// TwinCAT 3 PLC project CNC
// ProgramVersion: 3.1.4020.2
// libraries:
//   Tc2_ControllerToolbox, * (Beckhoff Automation GmbH)
//   Tc2_MC2, * (Beckhoff Automation GmbH)
//   Tc2_Standard, * (Beckhoff Automation GmbH)
//   Tc2_System, * (Beckhoff Automation GmbH)
//   Tc2_TcpIp, * (Beckhoff Automation GmbH)
//   Tc3_Interfaces, * (Beckhoff Automation GmbH)
//   Tc3_Module, * (Beckhoff Automation GmbH)
//   VisuDialogs, * (System)
// project tree:
//   DUTs/ E_ModeMMA.TcDUT, ST_Param.TcDUT, ST_ParamFixed.TcDUT, ST_ParamMachine.TcDUT, ST_ParamRecipe.TcDUT, ST_ParamStatus.TcDUT
//   DUTs/Param/ ST_Palette.TcDUT, ST_Position.TcDUT
//   / ErrorList.TcTLO, GlobalImagePool.TcGIPO (not stored), GlobalTextList.TcGTLO, PlcTask.TcTTO, Visualisierungsmanager.TcVMO (not stored), VISU_TASK.TcTTO
//   FB_Lib/Conversion/ FB_ConfigAnalog.TcPOU, FB_Ia.TcPOU, FB_Qa.TcPOU, ST_MinMax.TcDUT
//   FB_Lib/FB_ActionneurSimple/ FB_ActionneurSimple.TcPOU, ST_Erreur.TcDUT, ST_ParamActionneur.TcDUT
//   FB_Lib/ FB_Etape.TcPOU, FB_RegulMoteur.TcPOU (excluded from build)
//   FB_Lib/FB_GestionModes/ FB_Btn.TcPOU, FB_CycleAuto.TcPOU, FB_CycleInit.TcPOU, FB_CycleMan.TcPOU, FB_MMA.TcPOU, p_InitVar.TcPOU
//   FB_Lib/FB_GestionModes/IO/ ST_IO.TcDUT, ST_IOInput.TcDUT, ST_IOInputSimul.TcDUT, ST_IOOutput.TcDUT, ST_IOOutputSimul.TcDUT
//   FB_Lib/Motor/ FB_Moteur.TcPOU, ST_ParamMoteur.TcDUT, ST_ParamMoveMoteur.TcDUT
//   FB_Lib/TCPIP/ FB_TCP.TcPOU, ST_Output.TcDUT, ST_ParamTCP.TcDUT, ST_TxRx.TcDUT
//   GVLs/ GVL.TcGVL
//   POUs/ MAIN.TcPOU
//   VISUs/ Visu2_MainCtr.TcVIS, Visu2_LanguageUser.TcVIS, Visu2_Status.TcVIS, Visu2_StatusSimple.TcVIS, VisuAdmin.TcVIS, Visualization.TcVIS, VisuAuto.TcVIS, VisuInit.TcVIS, VisuManual.TcVIS, VisuMMA.TcVIS, VisuMotor.TcVIS (excluded from build)
// real-time tasks:
//   TASK PlcTask: cycle T#10ms, priority 10, ADS port 351
//   TASK VISU_TASK: cycle T#50000us, priority 12, ADS port 350
// motion (NC):
//   TASK NC-Task 1 SAF: cycle T#2ms, priority 4, ADS port 501
//   TASK NC-Task 1 SVB: cycle T#10ms, priority 8, ADS port 511
//   AXIS Axis 1 (id 1)
//     Dynamic: Acceleration=60900.1, Deceleration=60900.1, Jerk=1431970
//     Velo: RefSync=10, SlowManual=25, FastManual=3500, Maximum=3500
//     OtherSettings: AllowMotionCmdToSlave=true
//     encoder EncType=25
//       EncPara: ScaleFactorNumerator=360, ScaleFactorDenominator=12800, MaxCount=#x0000ffff
//         SoftEndMinControl: Enable=true
//         SoftEndMaxControl: Enable=true, Range=5000
//     drive DrvType=20
//       Analog: VeloReferenz=3500
//       TimeComp: TaskDelayCycles=1
//     controller CtrType=1
//       CtrPara: PriorControlFactor=1
//         PosDiffControl: Enable=false
//         PID: PosKp=60
//         Observer: BandWidth=20
//   AXIS Achse 2 - Y (id 2)
//     General: UnitName=°
//     Dynamic: Acceleration=127260, Deceleration=127260, Jerk=25706400
//     Velo: RefSearch=500, RefSync=100, SlowManual=20, FastManual=40000, Maximum=58000
//     TargetPosControl: Range=10
//     OtherSettings: AllowMotionCmdToSlave=true
//     encoder EncType=26
//       EncPara: ScaleFactorNumerator=360, ScaleFactorDenominator=2048, MaxCount=#x0000ffff
//         SoftEndMinControl: Enable=true
//         SoftEndMaxControl: Enable=true, Range=5000
//     drive DrvType=21
//       Analog: VeloReferenz=58000
//       TimeComp: TaskDelayCycles=1
//     controller CtrType=3
//       CtrPara: PriorControlFactor=1
//         PosDiffControl: Enable=false
//         PID: PosKp=30, PosTn=0.2, PosTv=0.2, PosTd=0.2, PosIOutputLimit=0.25, PosDOutputLimit=0.25
//         Observer: BandWidth=20
//   AXIS Achse 3 - Z (id 3)
//     Dynamic: Acceleration=3611.11, Deceleration=3611.11, Jerk=117362
//     Velo: Maximum=3500
//     OtherSettings: AllowMotionCmdToSlave=true
//     encoder EncType=1
//       EncPara: ScaleFactorNumerator=360, ScaleFactorDenominator=12600
//         SoftEndMinControl: Enable=true
//         SoftEndMaxControl: Enable=true, Range=125
//     drive DrvType=5
//       Analog: VeloReferenz=3500
//       TimeComp: TaskDelayCycles=1
//     controller CtrType=1
//       CtrPara: PriorControlFactor=1
//         PosDiffControl: Enable=false
//         PID: PosKp=60
//         Observer: BandWidth=20
// I/O:
//   DEVICE Gerät 2 (EtherCAT)
//     Box 1 (BK1150)
//     Box 2 (BK1150) (disabled)
// variable links:
//   NC-Task 1 SAF/Axes/Achse 2 - Y <-> Device 2 (EtherCAT)/Box 1 (BK1150)
//     Drive/Inputs/In/nState1 @bit 4 <-> Term 4 (KL2552)/Channel 1/Status @bit 4
//     Drive/Outputs/Out/nCtrl1 @bit 5 <-> Term 4 (KL2552)/Channel 1/Kontrolle @bit 5
//     Drive/Outputs/Out/nDataOut2[0] <-> Term 4 (KL2552)/Channel 1/Daten Aus
//     Enc/Inputs/In/nDataIn1[0] <-> Term 4 (KL2552)/Channel 1/Daten Ein
//     Enc/Inputs/In/nState1 @bit 2 <-> Term 4 (KL2552)/Channel 1/Status
//     Enc/Outputs/Out/nCtrl1 @bit 1 <-> Term 4 (KL2552)/Channel 1/Kontrolle
//   NC-Task 1 SAF/Axes/Axis 1 <-> Device 2 (EtherCAT)/Box 1 (BK1150)
//     Drive/Inputs/In/nState1 <-> Term 3 (KL2531)/Channel 1/Status
//     Drive/Outputs/Out/nCtrl1 <-> Term 3 (KL2531)/Channel 1/Ctrl
//     Drive/Outputs/Out/nDataOut2[0] <-> Term 3 (KL2531)/Channel 1/Velocity
//     Enc/Inputs/In/nDataIn1[0] <-> Term 3 (KL2531)/Channel 1/Position
//     Enc/Inputs/In/nState1 <-> Term 3 (KL2531)/Channel 1/ExtStatus
//     Enc/Outputs/Out/nCtrl1 <-> Term 3 (KL2531)/Channel 1/ExtCtrl
//   CNC/CNC Instance <-> Device 2 (EtherCAT)/Box 1 (BK1150)
//     PlcTask Inputs/GVL.fbAct1.IxSensIn <-> Term 7 (KL1408)/Channel 2/Eingang
//     PlcTask Inputs/GVL.fbAct1.IxSensOut <-> Term 7 (KL1408)/Channel 1/Eingang
//     PlcTask Inputs/GVL.stIO.stIn.IxAruIO <-> Term 8 (KL1408)/Channel 1/Eingang
//     PlcTask Inputs/GVL.stIO.stIn.xAirPressureOk <-> Term 8 (KL1408)/Channel 4/Eingang
//     PlcTask Inputs/GVL.stIO.stIn.xAllowedGetPiece <-> Term 7 (KL1408)/Channel 6/Eingang
//     PlcTask Inputs/GVL.stIO.stIn.xPiecePresent <-> Term 7 (KL1408)/Channel 7/Eingang
//     PlcTask Outputs/GVL.fbAct1.QxBlockingValve <-> Term 10 (KL2408)/Channel 2/Ausgang
//     PlcTask Outputs/GVL.fbAct1.QxInOutput <-> Term 9 (KL2408)/Channel 6/Ausgang
//     PlcTask Outputs/GVL.fbAct1.QxOutOutput <-> Term 9 (KL2408)/Channel 5/Ausgang
//     PlcTask Outputs/GVL.stIO.stOut.QxLampeOrange <-> Term 9 (KL2408)/Channel 2/Ausgang
//     PlcTask Outputs/GVL.stIO.stOut.QxLampeRed <-> Term 9 (KL2408)/Channel 1/Ausgang
//     PlcTask Outputs/GVL.stIO.stOut.QxLampeVerte <-> Term 9 (KL2408)/Channel 3/Ausgang
//   CNC/CNC Instance <-> NC-Task 1 SAF/Axes/Achse 2 - Y
//     PlcTask Inputs/GVL.fbMotorY.fbAxisRef.NcToPlc <-> Outputs/ToPlc
//     PlcTask Outputs/GVL.fbMotorY.fbAxisRef.PlcToNc <-> Inputs/FromPlc
//   CNC/CNC Instance <-> NC-Task 1 SAF/Axes/Achse 3 - Z
//     PlcTask Inputs/GVL.fbMotorZ.fbAxisRef.NcToPlc <-> Outputs/ToPlc
//     PlcTask Outputs/GVL.fbMotorZ.fbAxisRef.PlcToNc <-> Inputs/FromPlc
//   CNC/CNC Instance <-> NC-Task 1 SAF/Axes/Axis 1
//     PlcTask Inputs/GVL.fbMotorX.fbAxisRef.NcToPlc <-> Outputs/ToPlc
//     PlcTask Outputs/GVL.fbMotorX.fbAxisRef.PlcToNc <-> Inputs/FromPlc

CONFIGURATION CNC
    RESOURCE PLC ON TwinCAT3
        TASK PlcTask(INTERVAL := T#10ms, PRIORITY := 10);
        TASK VISU_TASK(INTERVAL := T#50000us, PRIORITY := 12);
        PROGRAM MAIN WITH PlcTask : MAIN;
        PROGRAM VisuElems_Visu_Prg WITH VISU_TASK : VisuElems.Visu_Prg;
    END_RESOURCE
END_CONFIGURATION

// ---- DUTs/E_ModeMMA.TcDUT

TYPE E_ModeMMA :
(
	Init := 0,
	Auto,
	Man
);
END_TYPE

// ---- DUTs/Param/ST_Palette.TcDUT
TYPE ST_Palette :
STRUCT
	PaletteDimensionX : INT;
	PaletteDimensionY : INT;
	
	ActualPalettePositionX : INT;
	ActualPalettePositionY : INT;
END_STRUCT
END_TYPE

// ---- DUTs/Param/ST_Position.TcDUT
TYPE ST_Position :
STRUCT
	PosX : LREAL;
	PosY: LREAL;
	Initialized: BOOL;
END_STRUCT
END_TYPE

// ---- DUTs/ST_Param.TcDUT
TYPE ST_Param :
STRUCT
	stStatus:ST_ParamStatus;	//informations d'états (compteur de pièces, modes,...)
	stFixed:ST_ParamFixed;		//Paramètres pas en lien avec le produit, fixe
	stRecipe:ST_ParamRecipe;	//Paramètres en lien avec le produit
	stMachine:ST_ParamMachine;	//Parametres de la machine
END_STRUCT
END_TYPE

// ---- DUTs/ST_ParamFixed.TcDUT
TYPE ST_ParamFixed :
STRUCT
END_STRUCT
END_TYPE

// ---- DUTs/ST_ParamMachine.TcDUT
TYPE ST_ParamMachine :
STRUCT
	stParamMotX:ST_ParamMoteur;		//parametres des trois Moteurs
	stParamMotY:ST_ParamMoteur;
	stParamMotZ:ST_ParamMoteur;
	
	stPosition0: ST_Position;		//Position Home
	stPosition1: ST_Position;		//Position Palette bottom left
	stPosition2: ST_Position;		//Position Palette bottom right
	stPosition3: ST_Position;		//Position Palette top left
	stPosition4: ST_Position;		//Position Prise Piece


END_STRUCT
END_TYPE

// ---- DUTs/ST_ParamRecipe.TcDUT
TYPE ST_ParamRecipe :
STRUCT
	stPalette1 : ST_Palette;
END_STRUCT
END_TYPE

// ---- DUTs/ST_ParamStatus.TcDUT
TYPE ST_ParamStatus :
STRUCT
	eMMA : E_ModeMMA; 
	xModePasAPas:BOOL;
	xErreur:BOOL;		//shows the current error state
	iId : INT; 			//error number currently active
	sMessage : STRING; 	//error message for the active error
	xInitOk:BOOL;		//indique que l'initialisation a été exécutée
	xHomingDone : BOOL;	//indique q'on a fait un homing depuis la derniere mise en puissance
END_STRUCT
END_TYPE

// ---- FB_Lib/Conversion/ST_MinMax.TcDUT
TYPE ST_MinMax :
STRUCT
	lrMin: LREAL;
	lrMax: LREAL;
END_STRUCT
END_TYPE

// ---- FB_Lib/FB_ActionneurSimple/ST_Erreur.TcDUT
TYPE ST_Erreur :
STRUCT
	xState:BOOL; 		//shows the current error state
	iId : INT; 			//error number currently active
END_STRUCT
END_TYPE

// ---- FB_Lib/FB_ActionneurSimple/ST_ParamActionneur.TcDUT
TYPE ST_ParamActionneur :
STRUCT
	tTimeOut : TIME; 			//max time allowed for moving to position bevor xState=TRUE
	xPresenceSensOut : BOOL; 	//If at the out-pos a Sensor is available
	xPresenceSensIn : BOOL; 	//If at the in-pos a Sensor is availaible
	tMoveOutTimeDelay : TIME; 	//delay after activating xPresenceSensOut before turning off output. When there is no Sensor, only this time will be used.
	tMoveInTimeDelay : TIME; 	//delay after activating xPresenceSensIn before turning off output. When there is no Sensor, only this time will be used.
END_STRUCT
END_TYPE

// ---- FB_Lib/FB_GestionModes/IO/ST_IO.TcDUT
TYPE ST_IO :
STRUCT
	stIn:ST_IOInput;
	stOut:ST_IOOutput;
END_STRUCT
END_TYPE

// ---- FB_Lib/FB_GestionModes/IO/ST_IOInput.TcDUT
TYPE ST_IOInput :
STRUCT
	IxAruIO AT%I*  :BOOL;
	xStartIO AT%I* :BOOL;
	xStopIO AT%I*  :BOOL;
	xResetIO AT%I* :BOOL;
	xAuto AT%I* : BOOL;
	xManual AT%I* : BOOL;
	
	
	
	iSetSpeedMotor : INT := 10;
	
	xAirPressureOk AT%I* : BOOL;
	
	//Btn in manual mode
	xHomingPosReached AT%I* : BOOL;
	xManualAct1GoIn AT%I* : BOOL;
	xManualAct1GoOut AT%I* : BOOL;
	
	//Btn in init mode
	xSetHomePos   AT%I*: BOOL;
	xJogXForward  AT%I*: BOOL;
	xJogYForward  AT%I*: BOOL;
	xJogXBackward AT%I*: BOOL;
	xJogYBackward AT%I*: BOOL;
	
	//Auto mode
	xAllowedGetPiece AT%I* : BOOL;
	xPiecePresent AT%I* : BOOL;
	xEmulateZDone AT%I* :Bool;
	
END_STRUCT
END_TYPE

// ---- FB_Lib/FB_GestionModes/IO/ST_IOInputSimul.TcDUT
TYPE ST_IOInputSimul :
STRUCT
	IxAru :BOOL;
END_STRUCT
END_TYPE

// ---- FB_Lib/FB_GestionModes/IO/ST_IOOutput.TcDUT
TYPE ST_IOOutput :
STRUCT
	QxLampeRed AT%Q*:BOOL;
	QxLampeVerte AT%Q* : BOOL;
	QxLampeOrange AT%Q* :BOOL;
	
	
END_STRUCT
END_TYPE

// ---- FB_Lib/FB_GestionModes/IO/ST_IOOutputSimul.TcDUT
TYPE ST_IOOutputSimul :
STRUCT
	QxLampeRed AT%Q*:BOOL;
END_STRUCT
END_TYPE

// ---- FB_Lib/Motor/ST_ParamMoteur.TcDUT
TYPE ST_ParamMoteur :
STRUCT
	stMoveLent:ST_ParamMoveMoteur;//paramètre déplacement lent
	stMoveRapide:ST_ParamMoveMoteur;//paramètre déplacement rapide
	lrPositionInitiale:LREAL:=0;//valeur de position initiale après un MC_Home;
	mcHomingMode:MC_HomingMode:=MC_Direct;//type homing
	(*HomingMode determines in which way the calibration is carried out.
    MC_DefaultHoming
    Initiates standard homing.
    MC_Direct
    Sets the axis position directly to Position without executing a movement.
    MC_ForceCalibration
    Enforces the "axis is calibrated" state. No movement takes place, and the position remains unchanged.
    MC_ResetCalibration
    Resets the calibration state of the axis. No movement takes place, and the position remains unchanged.*)
END_STRUCT
END_TYPE

// ---- FB_Lib/Motor/ST_ParamMoveMoteur.TcDUT
TYPE ST_ParamMoveMoteur :
STRUCT
	lrVitesse:LREAL:=900;			//vitesse
	lrAcceleration:LREAL:=0;		//accélération standard, 0 si standard
	lrDecceleration:LREAL:=0;		//accélération standard, 0 si standard
END_STRUCT
END_TYPE

// ---- FB_Lib/TCPIP/ST_Output.TcDUT
TYPE ST_Output :
STRUCT
	xBusy: BOOL;
	xError: BOOL;
	nErrID : INT;
	Resulte : STRING;
	Resulth : STRING;
	Resultd : STRING;
	Boole : INT;
	Boolh : INT;
	Boold : INT;
END_STRUCT
END_TYPE

// ---- FB_Lib/TCPIP/ST_ParamTCP.TcDUT
TYPE ST_ParamTCP :
STRUCT
	sRemoteHost : T_IPV4Addr;
	nRemotePort : UDINT;
	tTimeout: TIME;
	xConnected : BOOL;			//TRUE if currently Connected to a Server
	hSocket : T_HSOCKET;		//saves the connection details after the first Connection
	xCognexMode : BOOL;			//login in into an cognex Camera
	sCognexUser: STRING;
	sCognexPW: STRING;
	xConnectedCognex: BOOL;		//connection to Cognex etablished
	NetID :  T_AmsNetId;
END_STRUCT
END_TYPE

// ---- FB_Lib/TCPIP/ST_TxRx.TcDUT
TYPE ST_TxRx :
STRUCT
	sSend : STRING;
	sReceived: STRING;
END_STRUCT
END_TYPE

// ---- GVLs/GVL.TcGVL
VAR_GLOBAL

	fbAct1:FB_ActionneurSimple;	//Act1 corresponds to holding the object
	
	xModeStepForStep :BOOL;
	xNextStep : BOOL;
	
	//pour FB_gestion du mode
	fbMMA:FB_MMA;
	fbCycleAuto:FB_CycleAuto;
	fbCycleInit : FB_CycleInit;
	fbCycleMan : FB_CycleMan;
	
	stParam:ST_Param;
	fbBtn:FB_Btn;
	stIO:ST_IO;
	
	//Tachymetre moteur
	//fbMotor : FB_RegulMoteur;
	fbMotorX : FB_Moteur;
	fbMotorY : FB_Moteur;
	fbMotorZ : FB_Moteur;
	

	 
END_VAR

// ---- POUs/MAIN.TcPOU
PROGRAM MAIN
VAR
END_VAR

//******************************************
//cyclic call of all needed FB
//******************************************
ACT_Moteur();
ACT_Actor();

fbMMA();

//copy physical Inputs in fbBtn
fbBtn.xAru:=stio.stIn.IxAruIO;
fbBtn.xReset:=stio.stIn.xResetIO OR NOT stio.stIn.xAirPressureOk;
fbBtn.xStart:=stio.stIn.xStartIO;
fbBtn.xStop:=stio.stIn.xStopIO;
fbBtn.xAirPressureOk:=stio.stIn.xAirPressureOk;
fbBtn.xManualAct1GoIn:=stio.stIn.xManualAct1GoIn;
fbBtn.xManualAct1GoOut:=stio.stIn.xManualAct1GoOut;
fbBtn.xHomingPosReached:=stio.stIn.xHomingPosReached;
fbBtn.xSetHomePos:=stio.stIn.xSetHomePos;
fbBtn.xAllowedGetPiece:=stio.stIn.xAllowedGetPiece;
fbBtn.xPiecePresent:=stio.stIn.xPiecePresent;
fbBtn.xEmulateZDone:=stio.stIn.xEmulateZDone;
fbBtn.xJogXBackward:=stio.stIn.xJogXBackward;
fbBtn.xJogYBackward:=stio.stIn.xJogYBackward;
fbBtn.xJogXForward:=stio.stIn.xJogXForward;
fbBtn.xJogYForward:=stio.stIn.xJogYForward;
fbBtn.iMotorSpeed:=stio.stIn.iSetSpeedMotor;


//and now call it
fbBtn();

//stParam
//check for active errors
IF (fbAct1.stError.xState) THEN
	stParam.stStatus.xErreur:=TRUE;
	stParam.stStatus.iId:=fbAct1.stError.iId;
ELSIF (fbCycleAuto.xError) THEN
	stParam.stStatus.xErreur:=TRUE;
	stParam.stStatus.iId:=fbCycleAuto.iId;
ELSIF NOT fbBtn.xAirPressureOk THEN
	stParam.stStatus.xErreur:=TRUE;
	stParam.stStatus.iId:=1;
ELSE
	//clear the error State. Do not clear the last error Message to have some kind of error history
	stParam.stStatus.xErreur:=FALSE;
END_IF

//call auto mode and give over the needed parameters
fbCycleAuto.xStart:=fbMMA.iEtape=350;
fbCycleAuto.xStop:= fbMMA.iEtape=390;
fbCycleAuto.xReset:= fbMMA.iEtape=810 OR fbMMA.iEtape=910;
fbCycleAuto();

//call Init mode and give over the needed parameters
fbCycleInit.xStart:=(fbMMA.iEtape=110 OR fbMMA.iEtape=340);
fbCycleInit.xStop:= NOT (fbMMA.iEtape=111 OR fbMMA.iEtape=341);
fbCycleInit.xReset:= fbMMA.iEtape=810 OR fbMMA.iEtape=910;
fbCycleInit();
	
//call Manual mode and give over the needed parameters
fbCycleMan.xStart:= fbMMA.iEtape=210;
fbCycleMan.xStop:=  fbMMa.iEtape<>210;
fbCycleMan();


//******************************************
//Output actions
//******************************************

//activate Lamp1
stIo.stOut.QxLampeRed:=NOT fbBtn.xAru;

ACTION ACT_Actor:
//Air-Actor controlling part
//cyclic call of the FB-blocs
fbAct1();	//Act2 corresponds to taking the object

//actuator movement autorize only if not in ARU
fbAct1.xAutorizeIn:=fbBtn.xAru;
fbAct1.xAutorizeOut:=fbBtn.xAru;

//move in and out each actuator
fbAct1.xInGoOut:=fbCycleAuto.iEtape=113 OR fbCycleMan.iEtape=202;

fbAct1.xInGoIn:=fbCycleAuto.iEtape=180 OR fbCycleAuto.iEtape=122 OR fbCycleAuto.iEtape=150 OR fbCycleAuto.iEtape=800 OR fbCycleInit.iEtape=400 OR fbCycleMan.iEtape=201;

//Reset des Actionneurs avan le init
fbAct1.xReset:=fbCycleInit.iEtape=99 OR fbMMA.iEtape=810;
END_ACTION

ACTION ACT_Moteur:
//Motor controlling part
//exécution de l'appel du bloc moteur
fbMotorX(stParam:=stParam.stMachine.stParamMotX);
fbMotorY(stParam:=stParam.stMachine.stParamMotY);
fbMotorZ(stParam:=stParam.stMachine.stParamMotZ);


//pilotage mise en puissance
fbMotorX.mcPower.Enable:=stIO.stIn.IxAruIO;
fbMotorX.mcPower.Enable_Negative:=stIO.stIn.IxAruIO;
fbMotorX.mcPower.Enable_positive:=stIO.stIn.IxAruIO;
fbMotorX.mcPower.Override:=fbBtn.iMotorSpeed;
fbMotorX.mSetMoveAbsRapide();

fbMotorY.mcPower.Enable:=stIO.stIn.IxAruIO;
fbMotorY.mcPower.Enable_Negative:=stIO.stIn.IxAruIO;
fbMotorY.mcPower.Enable_positive:=stIO.stIn.IxAruIO;
fbMotorY.mcPower.Override:=fbBtn.iMotorSpeed;
fbMotorY.mSetMoveAbsLent();

fbMotorZ.mcPower.Enable:=stIO.stIn.IxAruIO;
fbMotorZ.mcPower.Enable_Negative:=stIO.stIn.IxAruIO;
fbMotorZ.mcPower.Enable_positive:=stIO.stIn.IxAruIO;
fbMotorZ.mcPower.Override:=fbBtn.iMotorSpeed;
fbMotorY.mSetMoveAbsLent();


//pilotage homing (prise d'origine)
fbMotorX.mcHome.Execute:=fbCycleInit.iEtape=100;
fbMotorX.mcHome.bCalibrationCam:=fbBtn.xHomingPosReached;

//pilotage homing (prise d'origine)
fbMotorY.mcHome.Execute:=fbCycleInit.iEtape=200;
fbMotorY.mcHome.bCalibrationCam:=fbBtn.xHomingPosReached;

//pilotage homing (prise d'origine)
fbMotorZ.mcHome.Execute:=fbCycleInit.iEtape=300;
fbMotorZ.mcHome.bCalibrationCam:=fbBtn.xHomingPosReached;


//pilotage Rest
fbMotorX.mcReset.Execute:=fbMMA.iEtape=810 OR fbCycleInit.iEtape=100;
fbMotorY.mcReset.Execute:=fbMMA.iEtape=810 OR fbCycleInit.iEtape=100;
fbMotorZ.mcReset.Execute:=fbMMA.iEtape=810 OR fbCycleInit.iEtape=100;

//pilotage déplacement absolu
fbMotorX.mcMoveAbsolute.Execute:=fbCycleAuto.iEtape=110 OR fbCycleAuto.iEtape=131;
fbMotorY.mcMoveAbsolute.Execute:=fbCycleAuto.iEtape=110 OR fbCycleAuto.iEtape=131;
fbMotorZ.mcMoveAbsolute.Execute:=fbCycleAuto.iEtape=112 OR fbCycleAuto.iEtape=120 OR fbCycleAuto.iEtape=141 OR fbCycleAuto.iEtape=161;

//Move Jog
fbMotorX.mcJog.JogForward:= fbBtn.xJogXForward AND (fbCycleInit.iEtape=500 OR fbCycleMan.iEtape=100);
fbMotorX.mcJog.JogBackwards:= fbBtn.xJogXBackward AND (fbCycleInit.iEtape=500 OR fbCycleMan.iEtape=100);
fbMotorY.mcJog.JogForward:= fbBtn.xJogYForward AND (fbCycleInit.iEtape=500 OR fbCycleMan.iEtape=100);
fbMotorY.mcJog.JogBackwards:= fbBtn.xJogYBackward AND (fbCycleInit.iEtape=500 OR fbCycleMan.iEtape=100);
END_ACTION

END_PROGRAM

// ---- FB_Lib/FB_ActionneurSimple/FB_ActionneurSimple.TcPOU
FUNCTION_BLOCK FB_ActionneurSimple
VAR_INPUT
	xInGoOut AT%I*:BOOL;				//input for going out
	xInGoIn AT%I*:BOOL;					//input for going in
	xReset AT%I*:BOOL;					//Reset all (go back to init state
	
	xAutorizeOut AT%I* : BOOL;			//allowed to do the move requested with xInGoOut, If this is false Programm will return an error
	xAutorizeIn AT%I* : BOOL;			//allowed to do the move requested with xInGoIn, If this is false Programm will return an error

	IxSensOut AT%I*:BOOL;				//Sensor for the reached In-Pos
	IxSensIn AT%I*:BOOL;				//Sensor for the reached Out-Pos
		
	stParam:ST_ParamActionneur;			//Param for actuator 
END_VAR
VAR_OUTPUT
	xInOutPos:BOOL;						//Actuator is in Out Position
	xInInPos:BOOL;						//Actuator is in In Position
	
	xGoingOutNow AT%Q*:BOOL; 			//indication that actor is going in Out-Pos
	xGoingInNow AT%Q*:BOOL; 			//indication that actor is going in In-Pos
	
	QxOutOutput AT%Q*:BOOL;				//Output to actuator for going Out
	QxInOutput AT%Q*:BOOL;				//Output to actuator for going In
	
	QxBlockingValve AT%Q* : BOOL; 		//Blocking valve. Only TRUE when autorisation is present.
										//TODO: put this in an external actuator
END_VAR
VAR
	fbEtape:FB_Etape;
	fbTimeOut:TON;
	fbRTrigOut:R_Trig;
	fbRTrigIn:R_Trig;
	
	stError:ST_Erreur;					//Error Struct

END_VAR

fbEtape.mActualisation(xModeStepForStep,xNextStep);

//check rising edges on 
fbRTrigOut(clk:=xInGoOut);
fbRTrigIn(clk:=xInGoIn);

//Go to the next step when there is an Out-Command
IF fbRTrigOut.Q AND NOT(fbEtape.iNo>=200 AND fbEtape.iNo<=299) THEN	//When rising-edge was detected
	IF xAutorizeOut THEN
		fbEtape.piVal:=200;
	ELSE
		stError.iId:=100;
	END_IF		
fbEtape.piVal:=200;	
END_IF

//Go to the next step when there is an In-Command
IF fbRTrigIn.Q AND NOT(fbEtape.iNo>=100 AND fbEtape.iNo<=199) THEN	//When rising-edge was detected and not already going In
	IF xAutorizeIn THEN
		fbEtape.piVal:=100;
	ELSE
		stError.iId:=101;
	END_IF	
END_IF

//Reset
IF xReset THEN
	fbEtape.piVal:=0;
	stError.xState:=0;
	xInOutPos:=0;
	xInInPos:=0;
END_IF

//check for blocking valve
QxBlockingValve:= (xAutorizeOut OR xAutorizeIn);

//reset error
IF stError.xState THEN
	stError.iId:=0;
END_IF


CASE fbEtape.iNo OF
	0:fbEtape.psMess:='Wait for an In or Out command';
	//************************************************
	100:fbEtape.psMess:='Action go In';
		IF xAutorizeIn THEN
			fbEtape.piVal:=110;
			fbEtape.tTimeQ:=stParam.tMoveInTimeDelay;
		END_IF
	110:fbEtape.psMess:='Going in, waiting for IxSensIn';
		IF (IxSensIn AND stParam.xPresenceSensIn) OR NOT stParam.xPresenceSensIn THEN
			fbEtape.piVal:=150;
		END_IF
	150:fbEtape.psMess:='Going in, waiting for Timer';
		IF fbEtape.xTimeQ THEN
			fbEtape.piSVal:=199;
		END_IF
	199:fbEtape.psMess:='In-Position reached';
		IF (NOT IxSensIn) AND stParam.xPresenceSensIn THEN
			fbEtape.piVal:=150;
		END_IF
	//****************************************************
	200:fbEtape.psMess:='Action go Out';
		IF xAutorizeOut THEN
			fbEtape.piVal:=210;
			fbEtape.tTimeQ:=stParam.tMoveInTimeDelay;
		END_IF
	210:fbEtape.psMess:='Going Out, waiting for IxSensOut';
		IF (IxSensOut AND stParam.xPresenceSensOut) OR NOT stParam.xPresenceSensOut THEN
			fbEtape.piVal:=250;
		END_IF
	250:fbEtape.psMess:='Going Out, waiting for Timer';
		IF fbEtape.xTimeQ THEN
			fbEtape.piSVal:=299;
		END_IF
	299:fbEtape.psMess:='Out-Pos reached';
		IF (NOT IxSensOut) AND stParam.xPresenceSensoUT THEN
			fbEtape.piVal:=250;
		END_IF
	
	999:fbEtape.psMess:='Error';
END_CASE

//Activation Timer
fbTimeOut(IN:=(fbEtape.iNo>100 AND fbEtape.iNo<199 OR fbEtape.iNo>200 AND fbEtape.iNo<299)
				AND (NOT fbRTrigIn.Q AND NOT fbRTrigOut.Q),PT:=stParam.tTimeOut);	


//stError.sMessage is not needed anymore. Only the ID is needed, to use it with a GlobalText List and have Multilangage Support
IF fbTimeOut.Q THEN
	IF fbEtape.iNo < 200 THEN
		stError.iId:=111;
	ELSIF fbEtape.iNo>200 THEN
		stError.iId:=110;
	END_IF
ELSIF IxSensIn AND IxSensOut THEN
	stError.iId:=120;
ELSIF xInGoOut AND xInGoIn THEN
	stError.iId:=121;
END_IF

stError.xState :=fbEtape.iNo=999 OR fbTimeOut.Q OR (IxSensIn AND IxSensOut) OR (xInGoIn AND xInGoOut);

//***********************************
//Output affectation
//***********************************

xInInPos:=fbEtape.iNo=199;
xInOutPos:=fbEtape.iNo=299;
xGoingInNow:= QxInOutput AND NOT IxSensIn;
xGoingOutNow:= QxOutOutput AND NOT IxSensOut;

QxOutOutput:=fbEtape.iNo>200 AND fbEtape.iNo<=299;
QxInOutput:=fbEtape.iNo>100 AND fbEtape.iNo<=199;

END_FUNCTION_BLOCK

// ---- FB_Lib/FB_Etape.TcPOU
FUNCTION_BLOCK FB_Etape
VAR_INPUT
	tTimeQ :TIME;			//Time to stay in one state after which xTimeQ will go to TRUE
END_VAR
VAR_OUTPUT
	tTimeState: TIME ; 		//passed time in the actual state
	xTimeQ : BOOL ;			//is TRUE when time passed in the actual State is greather then tTimeQ
	xTransition:BOOL; 		//information that the state has just changed. For use when entering a new State the first time
	iNo:INT:=0; 			//State number running at the moment
	sMess :STRING ; 		//Information message about the current running state
END_VAR
VAR
	iMemNo:INT;				//Used for xTransition. Saves the actual state of the machine
	fbTon:ton;				//Timer for the actual State
	fbRtrig:R_trig;			//detector for rising edges
	xMemModeStepByStep:BOOL;	//Mem for the actual running Mode (see method mActualisation)
	
END_VAR

//executed at each state-machine-loop
METHOD PUBLIC mActualisation
VAR_INPUT
	xModeStepByStep: BOOL; 		//activate the Stepping-Mode (TRUE=ON)
	xSetNextStep: BOOL; 		//go to the next Step on rising eddge
END_VAR
//manage StepByStep
//-----------------

//Detect rising edge
fbRtrig(CLK:=xSetNextStep);
//copy the mode input to use it in piSVal
xMemModeStepByStep:=xModeStepByStep;

//detect a state changement in the state machine
xTransition:=iNo<>iMemNo;

//start Method when the state has changed
IF xTransition THEN
	mTransition();
END_IF

//manage the Timer and associated Variabels
//-----------------------------------------
fbTON(IN:=(iNo=iMemNo), PT:=T#71582M47S295MS, ET=>tTimeState); //will be resetted when the state is changed

//going to TRUE when longer in the actual State than tTimeQ
xTimeQ:=(tTimeState>=tTimeQ);

//save the last running state
iMemNo:=iNo;
END_METHOD

//Executed when a State has changed
METHOD PRIVATE mTransition
//make a new String to display
sMess:=CONCAT('iNo:=',int_to_string(iNo));
END_METHOD

//going to the next step while paying attention to StepByStep Mode
PROPERTY PUBLIC piSVal : INT
SET
IF NOT xMemModeStepByStep THEN
	//Step by step mode is off
	iNo:=piSVal;
	ELSIF fbRtrig.Q THEN
		//a button press on "xSetNextStep" has been detected
		iNo:=piSVal;
END_IF
END_SET
END_PROPERTY

//going to the next step without paying attention to StepByStep Mode
PROPERTY PUBLIC piVal : INT
SET
//set the next step
iNo:=piVal;
END_SET
END_PROPERTY

//
PROPERTY PUBLIC psMess : STRING
SET
//write the description of the actual step to sMess
IF xTransition THEN
	sMess:=psMess;
END_IF
END_SET
END_PROPERTY

END_FUNCTION_BLOCK

// ---- FB_Lib/FB_GestionModes/FB_MMA.TcPOU
FUNCTION_BLOCK FB_MMA
VAR_OUTPUT
	iEtape:INT;
END_VAR
VAR
	fbEtape:FB_Etape;
	p_InitVar : p_InitVar;
END_VAR

fbEtape.mActualisation(FALSE,FALSE);

//activate ARU if system already running (fbEtape>10) and not in reset or already in ARU (fbEtape<800)
IF NOT fbBtn.xAru AND fbEtape.iNo>10 AND fbEtape.iNo<800 THEN
	fbEtape.piVal:=900; 
END_IF

//do reset
IF fbBtn.xReset AND fbEtape.iNo>10 AND fbEtape.iNo<800 THEN
	fbEtape.piVal:=800;
END_IF

CASE fbEtape.iNo OF
	0:fbEtape.psMess:='MMA | Booting MMA';
		fbEtape.piVal:=10;
	
	10:	fbEtape.psMess:='MMA | Init stock-Variables';
		//OB100 Siemens
		p_InitVar(); //initialiser les vars (propre a la machine)
		fbEtape.piVal:=50;
	
	50:fbEtape.psMess:='MMA | Selection du mode MMA';
		IF (stParam.stStatus.eMMA=Auto) THEN
			fbEtape.piVal:=300;
		ELSIF (stParam.stStatus.eMMA=Man) THEN
			fbEtape.piVal:=210;
		ELSIF (stParam.stStatus.eMMA=Init) THEN
			fbEtape.piVal:=100;
		END_IF
		
	//--------------------------------------------------------------
	//Init
	//--------------------------------------------------------------
	100:fbEtape.psMess:='MMA | Init | Wait for fbBtn.xStart';
		IF (fbBtn.xStart) THEN
			fbEtape.piVal:=110;
		ELSIF (stParam.stStatus.eMMA<>Init) THEN
			fbEtape.piVal:=50;
		END_IF
	110:fbEtape.psMess:='MMA | Init | Wait end';
		IF fbCycleInit.iEtape=999 THEN
		fbEtape.piVal:=50;
		END_IF
	111:fbEtape.psMess:='MMA | Init | Finished';
		IF fbCycleInit.xBusy THEN
		fbEtape.piVal:=50;
		END_IF
		
	//--------------------------------------------------------------
	//Manual
	//--------------------------------------------------------------
	210:fbEtape.psMess:='MMA | Manual | Wait for mode changing';
		IF (stParam.stStatus.eMMA<>Man) THEN
		fbEtape.piVal:=211;
		END_IF
	211:fbEtape.psMess:='MMA | Manual | Finishing';
		IF (fbCycleMan.xBusy) THEN
		fbEtape.piVal:=50;
		END_IF
		
	//--------------------------------------------------------------
	//Auto
	//--------------------------------------------------------------
	300:fbEtape.psMess:='MMA | Auto | Wait for fbBtn.xStart';
		IF fbBtn.xStart THEN
			fbEtape.piVal:=340;
		ELSIF (stParam.stStatus.eMMA<>Auto) THEN
			fbEtape.piVal:=50;
		END_IF
	
	340:fbEtape.psMess:='MMA | Auto | Do Init - Start';
		fbEtape.piVal:=341;
		
	341:fbEtape.psMess:='MMA | Auto | Do Init - Wait end';
		IF fbCycleInit.iEtape=999 THEN
			fbEtape.piVal:=350;
			stParam.stStatus.xInitOk:=TRUE;
		END_IF
		
	350:fbEtape.psMess:='MMA | Auto | Production - Wait Stop Signal';
		IF fbBtn.xStop THEN 
			fbEtape.piVal:=390;
		END_IF
		
	390:fbEtape.psMess:='MMA | Auto | Wait end';
		IF (NOT fbCycleAuto.xBusy) THEN
			fbEtape.piVal:=50;
		END_IF
		
	//--------------------------------------------------------------
	//Reset
	//--------------------------------------------------------------
	800:fbEtape.psMess:='MMA | Reset | Stopp all';
		fbEtape.piVal:=810;
	810:fbEtape.psMess:='MMA | Reset | Stopp all';
		fbEtape.piVal:=899;
	899:fbEtape.psMess:='MMA | Reset | Finished';
		IF fbBtn.xAirPressureOk THEN
			fbEtape.piVal:=50;
		END_IF
		
		
	//--------------------------------------------------------------
	//ARU
	//--------------------------------------------------------------
	900:fbEtape.psMess:='MMA | ARU | Stopp all';
		fbEtape.piVal:=910;
	910:fbEtape.psMess:='MMA | ARU | Stopp all';
		fbEtape.piVal:=950;
	950:fbEtape.psMess:='MMA | ARU | ok - Wait until resetting ARU-Btn';
		IF fbBtn.xAru THEN
			fbEtape.piVal:=999;
	END_IF
	999:fbEtape.psMess:='MMA | ARU | Finished';
		fbEtape.piVal:=50;
END_CASE

iEtape:=fbEtape.iNo;

END_FUNCTION_BLOCK

// ---- FB_Lib/FB_GestionModes/p_InitVar.TcPOU
FUNCTION_BLOCK p_InitVar
VAR_INPUT
END_VAR
VAR_OUTPUT
END_VAR
VAR
	tEnvStabSort: INT;
END_VAR

VisuElems.CURRENTLANGUAGE := 'de';

fbAct1.stParam.xPresenceSensIn:=TRUE;
fbAct1.stParam.xPresenceSensOut:=TRUE;
fbAct1.stParam.tTimeOut:=T#5S;
fbAct1.stParam.tMoveInTimeDelay:=T#0.2S;
fbAct1.stParam.tMoveOutTimeDelay:=T#0.2S;


stParam.stStatus.eMMA:=Init;

stParam.stMachine.stParamMotY.stMoveLent.lrVitesse:=4500;

stParam.stMachine.stParamMotX.stMoveRapide.lrVitesse:=3500;

stParam.stMachine.stParamMotZ.stMoveRapide.lrVitesse:=3500;
stParam.stMachine.stParamMotZ.stMoveLent.lrVitesse:=500;

//setup all reference positions. Except Position 0 cause this one needs to be calibrated
stParam.stMachine.stPosition1.Initialized:=TRUE;
stParam.stMachine.stPosition1.PosX:=1000;
stParam.stMachine.stPosition1.PosY:=1000;
stParam.stMachine.stPosition2.Initialized:=TRUE;
stParam.stMachine.stPosition2.PosX:=3000;
stParam.stMachine.stPosition2.PosY:=1000;
stParam.stMachine.stPosition3.Initialized:=TRUE;
stParam.stMachine.stPosition3.PosX:=1000;
stParam.stMachine.stPosition3.PosY:=3000;
stParam.stMachine.stPosition4.Initialized:=TRUE;
stParam.stMachine.stPosition4.PosX:=4000;
stParam.stMachine.stPosition4.PosY:=4000;

//setup the Palette
stParam.stRecipe.stPalette1.PaletteDimensionX:=10;
stParam.stRecipe.stPalette1.PaletteDimensionY:=10;

//init has not been done now
stParam.stStatus.xInitOk:=FALSE;
stParam.stStatus.xHomingDone:=FALSE;

END_FUNCTION_BLOCK

// ---- FB_Lib/FB_GestionModes/FB_CycleAuto.TcPOU
FUNCTION_BLOCK FB_CycleAuto
VAR_INPUT
	xStart:BOOL;
	xStop:BOOL;
	xReset:BOOL;
END_VAR
VAR_OUTPUT	
	xBusy:BOOL;
	xReady:BOOL;
	xError:BOOL;
	iEtape:INT;
	iId : INT; 			//error number currently active
	iNumberProduced : INT;
END_VAR
VAR
	fbEtape:FB_Etape;
	fbRtrigStart:R_trig;
	xMemStop:BOOL:=FALSE;		//Memorise the Stop-Flag
	fbMoteur: INT;
END_VAR

fbEtape.mActualisation(stParam.stStatus.xModePasAPas,fbBtn.xNextPas);

fbRtrigStart(clk:=xStart);

IF xStop THEN
	xMemStop:=TRUE;
END_IF

IF xReset THEN
	fbEtape.piVal:=0;
	xBusy:=FALSE;
END_IF

CASE fbEtape.iNo OF
	0:	fbEtape.psMess:='Auto | Start Cycle';
		IF fbRtrigStart.Q THEN
			xMemStop:=FALSE;
			fbEtape.piVal:=1;
			iNumberProduced:=0;
		END_IF
	1: fbEtape.psMess:='Auto | Check if initialized';
		IF  stParam.stMachine.stPosition0.Initialized AND stParam.stMachine.stPosition1.Initialized AND stParam.stMachine.stPosition2.Initialized AND stParam.stMachine.stPosition3.Initialized AND stParam.stMachine.stPosition4.Initialized THEN
			fbEtape.piSVal:=100;
		ELSE
			fbEtape.piSVal:=800;	
		END_IF
	100:fbEtape.psMess:='Auto | Wait UNTIL allowed TO go TO Pos4';
		IF fbBtn.xAllowedGetPiece THEN
			fbMotorX.mSetMoveAbsRapide();
			fbMotorX.mcMoveAbsolute.Position:=stParam.stMachine.stPosition0.PosX + stParam.stMachine.stPosition4.PosX;
			fbMotorY.mSetMoveAbsLent();
			fbMotorY.mcMoveAbsolute.Position:=stParam.stMachine.stPosition0.PosY + stParam.stMachine.stPosition4.PosY;
			fbEtape.piSVal:=110;
		ELSIF xMemStop=TRUE THEN
			fbEtape.piSVal:=999;
		END_IF		
	110:fbEtape.psMess:='Auto | Wait until in Pos 4';
		IF (fbMotorX.mcMoveAbsolute.Done AND fbMotorY.mcMoveAbsolute.Done) OR fbBtn.xEmulateZDone THEN
			fbEtape.piSVal:=111;
		END_IF
	111:fbEtape.psMess:='Auto | Putting down Z ';
		fbMotorZ.mSetMoveAbsLent();
		fbMotorZ.mcMoveAbsolute.Position:=100;
		fbEtape.piSVal:=112;
	112:fbEtape.psMess:='Auto | Waiting until Z is down';
		IF fbMotorZ.mcMoveAbsolute.Done OR fbBtn.xEmulateZDone THEN
			fbEtape.piSVal:=113;
		END_IF
	113:fbEtape.psMess:='Auto | Closing Act1';
		IF fbAct1.xInOutPos		THEN
			fbEtape.piVal:=120;
		END_IF
	120:fbEtape.psMess:='Auto | Z go up';
		fbMotorZ.mSetMoveAbsRapide();
		fbMotorZ.mcMoveAbsolute.Position:=0;
		fbEtape.piVal:=121; //all is ok;
	121:fbEtape.psMess:='Auto | Wait until Z is up and make a presence check';
		IF (fbMotorZ.mcMoveAbsolute.Done OR fbBtn.xEmulateZDone) AND fbBtn.xPiecePresent THEN
			fbEtape.piSVal:=130;
		END_IF
		IF (fbMotorZ.mcMoveAbsolute.Done OR fbBtn.xEmulateZDone) AND NOT fbBtn.xPiecePresent THEN
			fbEtape.piSVal:=122;
		END_IF
	122: fbEtape.psMess:='Auto | Open Act1 and go back one step';
		IF fbAct1.xInInPos THEN
			fbEtape.piSVal:=111;
		END_IF
	130:fbEtape.psMess:='Auto | Go back to palette position';
			//check and calculate Palette dimensions and position where to put the object
			IF stParam.stRecipe.stPalette1.ActualPalettePositionY >= stParam.stRecipe.stPalette1.PaletteDimensionY THEN
				stParam.stRecipe.stPalette1.ActualPalettePositionY :=0;
				stParam.stRecipe.stPalette1.ActualPalettePositionX := stParam.stRecipe.stPalette1.ActualPalettePositionX +1;
				IF stParam.stRecipe.stPalette1.ActualPalettePositionX >= stParam.stRecipe.stPalette1.PaletteDimensionX THEN
					fbEtape.piSVal:=800;		//nous sommes hors des butees de la palette
				END_IF
			END_IF
			//calculate X-Position. (Xmax-Xmin) / Nombre de pos en X = increment par positionX
			//						Xactualle*increments + XminPosition =Position de cible
			fbMotorX.mSetMoveAbsRapide();
			fbMotorX.mcMoveAbsolute.Position:=(stParam.stMachine.stPosition0.PosX + stParam.stMachine.stPosition1.PosX)
											+  stParam.stRecipe.stPalette1.ActualPalettePositionX
													* ( (stParam.stMachine.stPosition2.PosX-stParam.stMachine.stPosition0.PosX) / stParam.stRecipe.stPalette1.PaletteDimensionX );
			//meme chose pour Y
			fbMotorY.mSetMoveAbsLent();
			fbMotorY.mcMoveAbsolute.Position:=(stParam.stMachine.stPosition0.PosY + stParam.stMachine.stPosition1.PosY)
											+  stParam.stRecipe.stPalette1.ActualPalettePositionY
													* ( (stParam.stMachine.stPosition3.PosY-stParam.stMachine.stPosition0.PosY) / stParam.stRecipe.stPalette1.PaletteDimensionY );
			//increase the row number
			stparam.stRecipe.stPalette1.ActualPalettePositionY := 	stparam.stRecipe.stPalette1.ActualPalettePositionY +1;
			fbEtape.piSVal:=131;
	131:fbEtape.psMess:='Auto | Wait until in Pos 4';
		IF (fbMotorX.mcMoveAbsolute.Done AND fbMotorY.mcMoveAbsolute.Done) OR fbBtn.xEmulateZDone THEN
			fbEtape.piSVal:=140;
		END_IF
	140:fbEtape.psMess:='Auto | Putting down Z ';
		fbMotorZ.mSetMoveAbsLent();
		fbMotorZ.mcMoveAbsolute.Position:=100;
		fbEtape.piSVal:=141;
	141:fbEtape.psMess:='Auto | Waiting until Z is down';
		IF fbMotorZ.mcMoveAbsolute.Done OR fbBtn.xEmulateZDone THEN
			fbEtape.piSVal:=150;
		END_IF
	150:fbEtape.psMess:='Auto | Opening Act1';
		IF fbAct1.xInInPos		THEN
			fbEtape.piVal:=160;
		END_IF
	160:fbEtape.psMess:='Auto | Z go up';
		fbMotorZ.mSetMoveAbsRapide();
		fbMotorZ.mcMoveAbsolute.Position:=0;
		fbEtape.piVal:=161; //all is ok;
	161:fbEtape.psMess:='Auto | Wait until Z is up';
		IF  xMemStop=FALSE THEN
			fbEtape.piSVal:=100;
		ELSIF (fbMotorZ.mcMoveAbsolute.Done OR fbBtn.xEmulateZDone) AND xMemStop=TRUE THEN
			fbEtape.piSVal:=999;
		END_IF	
	
	800:fbEtape.psMess:='Auto | Error occured - Going into stock state';
		//turn off all motors and release all Actors
			fbEtape.piVal:=810;
	810:fbEtape.psMess:='Auto | Error occured - Press Reset to recover';
		//do nothing and wait
	
	999:fbEtape.psMess:='Auto | Finished';
		fbEtape.piVal:=0;
END_CASE

//***********************************
//Output affectation
//***********************************

xError:=(fbEtape.iNo=800 OR fbEtape.iNo=810);
xBusy:=fbEtape.iNo<>0;
xReady:=fbEtape.iNo=0;
iEtape:=fbEtape.iNo;

END_FUNCTION_BLOCK

// ---- FB_Lib/FB_GestionModes/FB_CycleInit.TcPOU
FUNCTION_BLOCK FB_CycleInit
VAR_INPUT
	xStart : BOOL;
	xStop : BOOL;
	xReset:BOOL;
END_VAR
VAR_OUTPUT
	fbRtrigStart:R_trig;
	xBusy:BOOL;
	iEtape:INT;
END_VAR
VAR
	fbEtape:FB_Etape;
END_VAR

fbEtape.mActualisation(stParam.stStatus.xModePasAPas,fbBtn.xNextPas);

fbRtrigStart(clk:=fbBtn.xStart);

IF xReset THEN
	fbEtape.piVal:=0;
	xBusy:=FALSE;
END_IF

CASE fbEtape.iNo OF
	0:fbEtape.psMess:='Init | Wait';
		IF xStart THEN
			fbEtape.piVal:=99;
		END_IF
	
	
	99: fbEtape.psMess:='Init | Reset on Actuators and Motor';
		IF  stParam.stStatus.xHomingDone=TRUE THEN
			fbEtape.piSVal:=400;
		ELSE
			fbEtape.piSVal:=100;
		END_IF
	100: fbEtape.psMess:='Start Homing X';
			fbEtape.tTimeQ:=T#100MS;
			fbEtape.piSVal:=101;
	101:fbEtape.psMess:='Init | Wait 100MS';
		IF fbEtape.xTimeQ THEN
			fbEtape.piSVal:=102;
		END_IF
	102: fbEtape.psMess:='Init | Waiting for Homing Axis X';
		IF NOT fbMotorX.mcHome.Active AND NOT fbBtn.xHomingPosReached THEN
			fbEtape.piVal:=200;
		END_IF
		
	200:fbEtape.psMess:='Init | Start Homing Axis Y';
		fbEtape.piVal:=201;
		fbEtape.tTimeQ:=T#100MS;
	201:fbEtape.psMess:='Init | Wait 100MS';
		IF fbEtape.xTimeQ THEN
			fbEtape.piSVal:=202;
		END_IF
	202: fbEtape.psMess:='Init | Waiting for Homing Axis Y';
		IF NOT fbMotorY.mcHome.Active AND NOT fbBtn.xHomingPosReached THEN
			fbEtape.piVal:=300;
		END_IF
		
	300:fbEtape.psMess:='Init | Start Homing Axis Z';
		fbEtape.piVal:=301;
		fbEtape.tTimeQ:=T#100MS;
	301:fbEtape.psMess:='Init | Wait 100MS';
		IF fbEtape.xTimeQ THEN
			fbEtape.piSVal:=302;
		END_IF
	302: fbEtape.psMess:='Init | Waiting for Homing Axis Z';
		IF NOT fbMotorZ.mcHome.Active AND NOT fbBtn.xHomingPosReached THEN
			fbEtape.piVal:=400;
			stParam.stStatus.xHomingDone:=TRUE;
		END_IF
		
		
	400:fbEtape.psMess:='Init | Init Actor1';
		IF  fbAct1.xInInPos AND stParam.stMachine.stPosition0.Initialized=FALSE THEN
			fbEtape.piSVal:=500;
		ELSIF  fbAct1.xInInPos AND stParam.stMachine.stPosition0.Initialized=TRUE THEN
			fbEtape.piSVal:=999;
		END_IF
		
	500:fbEtape.psMess:='Init | Init Home Position';
		IF  fbBtn.xSetHomePos THEN
			stParam.stMachine.stPosition0.Initialized:=TRUE;
			stParam.stMachine.stPosition0.PosX:=fbMotorX.fbAxisRef.NcToPlc.ActPos;
			stParam.stMachine.stPosition0.PosY:=fbMotorY.fbAxisRef.NcToPlc.ActPos;
			fbEtape.piSVal:=999;
		END_IF
		
		
	
	999:fbEtape.psMess:='Init | Finished';
		IF (xStop) THEN
		fbEtape.piSVal:=0;
	END_IF
END_CASE

xBusy:=fbEtape.iNo<>0;
iEtape:=fbEtape.iNo;

END_FUNCTION_BLOCK

// ---- FB_Lib/FB_GestionModes/FB_CycleMan.TcPOU
FUNCTION_BLOCK FB_CycleMan
VAR_INPUT
	xStart : BOOL;
	xStop : BOOL;
	
	
END_VAR
VAR_OUTPUT
	fbRtrigStart:R_trig;
	xBusy:BOOL;
	iEtape:INT;
END_VAR
VAR
	fbEtape:FB_Etape;
	inc: INT;
END_VAR

fbEtape.mActualisation(FALSE,FALSE);

fbRtrigStart(clk:=fbBtn.xStart);


CASE fbEtape.iNo OF
	0:	fbEtape.psMess:='Manual | Wait';
		IF xStart THEN
			fbEtape.piVal:=100;
		END_IF
	100:fbEtape.psMess:='Manual | Select what to do';
		//changer de mode
		IF  stParam.stStatus.eMMA<>Man THEN
			fbEtape.piSVal:=990;
		END_IF
		//Act1:
		IF (fbBtn.xManualAct1GoIn) THEN
			fbEtape.piVal:=201;
		END_IF
		IF (fbBtn.xManualAct1GoOut) THEN
			fbEtape.piVal:=202;
		END_IF
		IF fbBtn.xSetHomePos THEN
			fbEtape.piVal:=300;
		END_IF
		
		
		
		
	201: fbEtape.psMess:='Manual | Action : Act 1 Go in';
		IF (NOT fbBtn.xManualAct1GoIn) THEN
			fbEtape.piVal:=100;
		END_IF
	202: fbEtape.psMess:='Manual | Action : Act 1 Go out';
		IF (NOT fbBtn.xManualAct1GoOut) THEN
			fbEtape.piVal:=100;
		END_IF
	300: fbEtape.psMess:='Manual | Set Home Position';
		stParam.stMachine.stPosition0.Initialized:=TRUE;
		stParam.stMachine.stPosition0.PosX:=fbMotorX.fbAxisRef.NcToPlc.ActPos;
		stParam.stMachine.stPosition0.PosY:=fbMotorY.fbAxisRef.NcToPlc.ActPos;
		fbEtape.piVal:=100;
	
	990:fbEtape.psMess:='Manual | Finishing';
		//ici on fait des choses de fin (ex. eteindre un Motor qui tourne encore)
		IF (1) THEN
			fbEtape.piSVal:=999;
		END_IF	
	999:fbEtape.psMess:='Manual | Finished';
		IF (xStop) THEN
			fbEtape.piSVal:=0;
		END_IF
		
END_CASE

xBusy:=fbEtape.iNo<>0;
iEtape:=fbEtape.iNo;

END_FUNCTION_BLOCK

// ---- FB_Lib/FB_GestionModes/FB_Btn.TcPOU
FUNCTION_BLOCK FB_Btn
VAR_INPUT
	xStart:BOOL;
	xStop:BOOL;
	xReset:BOOL;
	xNextPas:BOOL;
	xAru:BOOL;
	xAirPressureOk : BOOL;
	iMotorSpeed: INT;
	
	//Auto mode
	xAllowedGetPiece: BOOL;
	xPiecePresent : BOOL;
	xEmulateZDone : BOOL;
	
	//Init Mode
	xHomingPosReached : BOOL;
	xJogXForward : BOOL;
	xJogXBackward: BOOL;
	xJogYForward : BOOL;
	xJogYBackward: BOOL;
	
	//Btn used in Manual-Mode
	xSetHomePos : BOOL;
	xManualAct1GoIn: BOOL;
	xManualAct1GoOut : BOOL;
END_VAR

END_FUNCTION_BLOCK

// ---- FB_Lib/FB_RegulMoteur.TcPOU
FUNCTION_BLOCK FB_RegulMoteur
VAR_INPUT
		Consigne: LREAL;					//sets the desired speed of the Motor in rot/min
		lrValeurDirection: LREAL;			//the converted value from Tachymeter with Direction added
		xDirection: BOOL;					//Forward or Backward
		xOnOff: BOOL;						//Motor On or Off
		PARA : ST_CTRL_PID_PARAMS;			//Parameters for the PID
		xReset: BOOL;						//Reset the PID-Block
		PID : FB_CTRL_PID;					//PID-Block
		fbConvertNumToMotorOut : FB_Qa;		//Convert the PID-Output into numeric values send to the motor
		fbConvertTachoToNumSpeed : FB_Ia;	//Convert the numeric values from the Tachymeter into rot/min
		TimerOffAlarm : UINT;				//after enabling the Motor all Alarms will be blocked for 2sec
END_VAR
VAR_OUTPUT
	xError : BOOL;							//Error state
	iErrorID : INT;							//Error ID
END_VAR

//convert Tacho speed into rot/min
fbConvertTachoToNumSpeed();

//call the PID-Block if needed
IF xOnOff THEN
	PID(fOut=>fbConvertNumToMotorOut.lrConsigne,fSetpointValue:=Consigne,
		fActualValue:=fbConvertTachoToNumSpeed.lrValeur,eMode:=2,stParams:=PARA);
	//decrese the delay for alarms
	IF TimerOffAlarm>0 THEN
		TimerOffAlarm:=TimerOffAlarm-1;
	END_IF
ELSE
	fbConvertNumToMotorOut.lrConsigne:=0;
	TimerOffAlarm:=200; //200 @ 10ms Cycle --> 2sec
END_IF

//Convert now to have the value as fast as possible written to the motor
fbConvertNumToMotorOut();

//Reset the PID block
IF xReset THEN
	PID.bSync:=xReset;
END_IF


//******************************************
//Output actions
//******************************************

//Error management
IF PID.bError AND xOnOff AND TimerOffAlarm=0 THEN
xError:=TRUE;
iErrorID:=300;
ELSIF PID.bARWactive AND xOnOff AND TimerOffAlarm=0 THEN
	xError:=TRUE;
	iErrorId:=301;
ELSE
	xError:=FALSE;
END_IF

END_FUNCTION_BLOCK

// ---- FB_Lib/Conversion/FB_Qa.TcPOU
FUNCTION_BLOCK FB_Qa
VAR_INPUT
	lrConsigne: LREAL;  		//user value to be converted in an analog value
	fbConfig: FB_ConfigAnalog; 	//Analog output configuration
END_VAR
VAR_OUTPUT
	QaSortie : DINT; 			//analog output
	lrEcart: LREAL; 			//actual error introduced while converting the value
	lrTension: LREAL; 			//Voltage on the Output-Pin depending on IrConsigne
END_VAR

//call the Method for converting
QaSortie:=fbConfig.mConvertValToAn(lrConsigne,lrTension=>lrTension,lrEcart=>lrEcart);

END_FUNCTION_BLOCK

// ---- FB_Lib/Conversion/FB_ConfigAnalog.TcPOU
FUNCTION_BLOCK FB_ConfigAnalog
VAR_INPUT
	uiNbreBitBus: UINT;		//resolution of the Bus in Bits
	(* revoir lequel des deux Bit... est vraiment utilisé *)
	uiNbreBitConv: UINT;	//resolution in bit of the AD-Converter 
	stTension: ST_minMax;	//max / min possible tension on the physical Pins
	stValeur: ST_minMax;	//max / min possible value in the user defined unit (ex. rot/min)
END_VAR
VAR
	udiNbreIncBus: UDINT;	//
	lrTemp: LREAL;			//
	lrValInc: LREAL;		//number of possible increments on the Bus
END_VAR

METHOD mCalculDelta : LREAL
VAR_INPUT
	stMinMax: ST_MinMax;
END_VAR
mCalculDelta:=stMinMax.lrMax-stMinMax.lrMin;
END_METHOD

METHOD mCalculInc : UDINT
VAR_INPUT
	uiNbreBitBus: UDINT;
END_VAR

mCalculInc:=SHL(1,uiNbreBitBus);
//mCaclulInc:=EXPT(2,uiNbreBitBus);
END_METHOD

METHOD mConvertAnToVal : LREAL
VAR_INPUT
	lrAna: LREAL; 		//RAW input value from the Analog Pin
END_VAR
VAR_OUTPUT
	///tension de la borne de sortie
	(* can this be removed ? *) lrTension: LREAL;
	///Ecart de l'escalier sur la borne de sortie en unité de valeur
	(* can this be removed ? *) lrEcart: LREAL;
	lrValeur: LREAL;	//Converted value in the user unit	
END_VAR
//Calculate number of increments
udiNbreIncBus:=mCalculInc(uiNbreBitBus);

//Start Converting
//apply a gain to the RAW input value
lrValeur:=0;	//réponse = 0 si hors condition
IF mCalculDelta(stValeur)<>0 THEN
	lrValeur:=(mCalculDelta(stValeur)/udiNbreIncBus)*lrAna;
END_IF

//Solution
mConvertAnToVal:=lrValeur;

(* are the following needed? *)
//Calculate the increment in the tension
lrEcart:=(mCalculDelta(stTension)/udiNbreIncBus);
//Solution in Voltage on the Input Pin
lrTension:=lrValInc*lrEcart+stTension.lrMin;
END_METHOD

METHOD mConvertValToAn : DINT
VAR_INPUT
	lrVal: LREAL;		//this is the setpoint value in the user unit
END_VAR
VAR_OUTPUT
	lrTension: LREAL;	//tension on the physical output pins
	lrEcart: LREAL;		//Error on the physical output
END_VAR
//Verfication if lrVal is really in the possible range set in stValeur
lrVal:=LIMIT(stValeur.lrMin,lrVal,stValeur.lrMax);

//Calculate the number of increments
udiNbreIncBus:=mCalculInc(uiNbreBitBus);

//Start Converting
//deltaTension/Nbreinc <-> deltaVal/Nbreinc val
lrTemp:=0;	//réponse = 0 si hors condition
IF mCalculDelta(stValeur)<>0 THEN
	//nombre d'incréments par rapport à lrVal, avec décalage de stValeur.lrMin
	lrValInc:=udiNbreIncBus*(lrVal-stValeur.lrMin)/mCalculDelta(stValeur);
	//décalage selon min max de la tension
	IF stTension.lrMin<0 THEN
		//ajout de l'offset si min négatif
		lrTemp:=lrValInc-udiNbreIncBus/2-1;
		ELSE
		lrTemp:=lrValInc;
	END_IF
END_IF
//résultat de la méthode
mConvertValToAn:=LREAL_TO_DINT(lrTemp);
//calcul de l'incrément tension
lrEcart:=(mCalculDelta(stTension)/udiNbreIncBus);
//résultat en unitée de tension
lrTension:=lrValInc*lrEcart+stTension.lrMin;
END_METHOD

END_FUNCTION_BLOCK

// ---- FB_Lib/Conversion/FB_Ia.TcPOU
FUNCTION_BLOCK FB_Ia
VAR_INPUT
	fbConfig: FB_ConfigAnalog;  //Analog Input configuration
	IaEntree: LREAL;			//Analog input value on the Input-Pin
END_VAR
VAR_OUTPUT
	lrValeur: LREAL; 			//converted value in the user unit
	(*Not used ? *)lrEcart: LREAL; 		///écart de précision sur la valeur de consigne => valeur +/- écart
	(*Not used ? *)lrTension: LREAL;	///tension en volt
END_VAR
VAR
END_VAR

//call the Method for converting
lrValeur:=fbConfig.mConvertAnToVal(IaEntree,lrTension=>lrTension,lrEcart=>lrEcart);

END_FUNCTION_BLOCK

// ---- FB_Lib/Motor/FB_Moteur.TcPOU
FUNCTION_BLOCK FB_Moteur
VAR_INPUT
	mcPower:MC_Power;					//mise ne puissance
	mcReset:MC_Reset;					//reset alarmes
	mcStop:MC_Stop;						//stop l'axe si en mouvement, après MC_Movevelocity
	mcHome:MC_Home;						//recherche de position initiale
	mcJog:MC_Jog;						//déplacemement en mode manuel
	mcMoveVelocity:MC_MoveVelocity;		//mise en vitesse
	mcMoveRelative:MC_MoveRelative;		//déplacement relatif
	mcMoveAbsolute:MC_MoveAbsolute;		//déplacement absolu
END_VAR
VAR_IN_OUT
	stParam:ST_ParamMoteur;
END_VAR
VAR_OUTPUT
	fbAxisRef:Axis_Ref;//lien avec le module NCPTP
	(*TYPE NCTOPLC_AXIS_REF
	STRUCT
	   StateDWord             : DWORD; (* Status double word *)
	   ErrorCode              : DWORD; (* Axis error code *)
	   AxisState              : DWORD; (* Axis moving status *)
	   AxisModeConfirmation   : DWORD; (* Axis mode confirmation (feedback from NC) *)
	   HomingState            : DWORD; (* State of axis calibration (homing) *)
	   CoupleState            : DWORD; (* Axis coupling state *)
	   SvbEntries             : DWORD; (* SVB entries/orders (SVB = Set preparation task) *)
	   SafEntries             : DWORD; (* SAF entries/orders (SAF = Set execution task) *)
	   AxisId                 : DWORD; (* Axis ID *)
	   OpModeDWord            : DWORD; (* Current operation mode *)
	   ActiveControlLoopIndex : WORD; (* Active control loop index *)
	   ControlLoopIndex       : WORD; (* Axis control loop index (0, 1, 2, when multiple control loops are used) *)
	   ActPos                 : LREAL; (* Actual position (absolut value from NC) *)
	   ModuloActPos           : LREAL; (* Actual modulo position *)
	   ModuloActTurns         : DINT; (* Actual modulo turns *)
	   ActVelo                : LREAL; (* Actual velocity *)
	   PosDiff                : LREAL; (* Position difference (lag distance) *)
	   SetPos                 : LREAL; (* Setpoint position *)
	   SetVelo                : LREAL; (* Setpoint velocity *)
	   SetAcc                 : LREAL; (* Setpoint acceleration *)
	   TargetPos              : LREAL; (* Estimated target position *)
	   ModuloSetPos           : LREAL; (* Setpoint modulo position *)
	   ModuloSetTurns         : DINT; (* Setpoint modulo turns *)
	   CmdNo                  : WORD; (* Continuous actual command number *)
	   CmdState               : WORD; (* Command state *)
	END_STRUCT
	END_TYPE*)
	xError:BOOL;//indique une erreur
END_VAR
VAR
END_VAR

mcPower(Axis:=fbAxisRef);
mcReset(Axis:=fbAxisRef);
mcStop(Axis:=fbAxisRef);
mcHome(Axis:=fbAxisRef);
mcJog(Axis:=fbAxisRef);
mcMoveVelocity(Axis:=fbAxisRef);
mcMoveRelative(Axis:=fbAxisRef);
mcMoveAbsolute(Axis:=fbAxisRef);
//refresh des status de moteur contenu dans fbAxisRef.Status
fbAxisRef.ReadStatus();

xError:=fbAxisRef.Status.Error
		OR mcPower.Error AND mcPower.Active 
		OR mcReset.Error AND mcReset.Execute
		OR mcStop.Error  AND mcStop.Active
		OR mcHome.Error  AND (mcHome.Execute OR mcHome.Active)
		OR mcJog.Error   AND (mcJog.JogBackwards OR mcJog.JogForward OR mcJog.Active)
		OR mcMoveVelocity.Error   AND (mcMoveVelocity.Execute OR mcMoveVelocity.Active)
		OR mcMoveRelative.Error  AND (mcMoveRelative.Execute OR mcMoveRelative.Active)
		OR mcMoveAbsolute.Error  AND (mcMoveAbsolute.Execute OR mcMoveAbsolute.Active);

METHOD mSetMoveAbsLent
VAR_INPUT
END_VAR
mcMoveAbsolute.Acceleration:=stParam.stMoveLent.lrAcceleration;
mcMoveAbsolute.Deceleration:=stParam.stMoveLent.lrDecceleration;
mcMoveAbsolute.Velocity:=stParam.stMoveLent.lrVitesse;
END_METHOD

METHOD mSetMoveAbsRapide
VAR_INPUT
END_VAR
mcMoveAbsolute.Acceleration:=stParam.stMoveRapide.lrAcceleration;
mcMoveAbsolute.Deceleration:=stParam.stMoveRapide.lrDecceleration;
mcMoveAbsolute.Velocity:=stParam.stMoveRapide.lrVitesse;
END_METHOD

END_FUNCTION_BLOCK

// ---- FB_Lib/TCPIP/FB_TCP.TcPOU
FUNCTION_BLOCK FB_TCP
VAR_INPUT
	xEnable : BOOL;					//true enables the communication and connect to host. False is like a reset: disconecting and disabling all Communication
	xForceDisconnect : BOOL;		//force a disconnect. Only needed when the Program starts the first time or when there is a Reset
	TxRx : ST_TxRx;					//Tx and Rx Strings
	TCPParam : ST_ParamTCP;			//Parameters for the Communication
	
	OutputDisconnect : ST_Output;	//Error and Output variales of each Method
	OutputDisconnectAll : ST_Output;
	OutputConnect : ST_Output;
	OutputSend : ST_Output;
	OutputReceive : ST_Output;

END_VAR
VAR_OUTPUT
	OutputGlobal : ST_Output;		//Global Error and Output struct
END_VAR
VAR
	fbConnect : FB_SocketConnect;		//for Method MConnect
	fbDisconnectAll : FB_SocketCloseAll;
	fbDisconnect : FB_SocketClose;
	FEdgeBusyConnect : F_Trig;
	REdge : R_Trig;	
	FEdge : F_Trig;
	
	fbReceive : FB_SocketReceive;		//for Method MReceive
	Timer : TON;
	xReceiveToFast: BOOL;
	sReceivedBuffer : STRING;
	
	fbSend : FB_SocketSend;				//for Method MSend
	fbRTrig:F_Trig;
	
	iCounter : INT;						//used in MCognex
END_VAR

mConnect();
mSend();
mReceive();
mCognex();

//******************************************
//Output actions
//******************************************

//Busy
OutputGlobal.xBusy:=OutputReceive.xBusy OR OutputSend.xBusy OR OutputConnect.xBusy OR OutputDisconnect.xBusy OR OutputDisconnectAll.xBusy;
//Errors
IF(OutputReceive.xError) THEN
	OutputGlobal.xError:=TRUE;
	OutputGlobal.nErrID:=OutputReceive.nErrID;
ELSIF (OutputSend.xError) THEN
	OutputGlobal.xError:=TRUE;
	OutputGlobal.nErrID:=OutputSend.nErrID;
ELSIF (OutputConnect.xError) THEN
	OutputGlobal.xError:=TRUE;
	OutputGlobal.nErrID:=OutputConnect.nErrID;
ELSIF (OutputDisconnect.xError) THEN
	OutputGlobal.xError:=TRUE;
	OutputGlobal.nErrID:=OutputDisconnect.nErrID;
ELSIF (OutputDisconnectAll.xError) THEN
	OutputGlobal.xError:=TRUE;
	OutputGlobal.nErrID:=OutputDisconnectAll.nErrID;
ELSE
	OutputGlobal.xError:=FALSE;
END_IF

METHOD PUBLIC mCognex
VAR
	TempPos1 : INT;
	TempPos2 : INT;
	
	Temp1: STRING;
	Temp2 : STRING;
	Temp3:STRING;
	
	
END_VAR
//etablish a Telnet-Connection to the Camera to communicate via the native Protocoll
IF TCPParam.xConnected AND TCPParam.xCognexMode THEN
	IF TxRx.sReceived='User: ' AND iCounter=0 THEN
		TxRx.sSend:='admin';
		iCounter:=1;
	END_IF
	IF TxRx.sReceived='Password: ' AND iCounter=1 THEN
		TxRx.sSend:='$R$N';
		iCounter:=2;
	END_IF
	IF TxRx.sReceived='User Logged In$R$N' AND iCounter=2 THEN
		TCPParam.xConnectedCognex:=TRUE;
	END_IF
END_IF

//when the camera sends the mesured data extract them from the String
IF TCPParam.xConnected AND TCPParam.xCognexMode THEN
	IF FIND(fbTCP.TxRx.sReceived,'PASS')>0 OR FIND(fbTCP.TxRx.sReceived,'FAIL')>0 THEN
		//The camera has send the string with the Mesurement results
		//extract mesured values
		TempPos1:=FIND(fbTCP.TxRx.sReceived, ';e:');
		TempPos2:=FIND(fbTCP.TxRx.sReceived, ';h:');
		OutputGlobal.Resulte:=MID(fbTCP.TxRx.sReceived,TempPos2-(TempPos1+3),TempPos1+3);
		
		TempPos1:=FIND(fbTCP.TxRx.sReceived, ';h:');
		TempPos2:=FIND(fbTCP.TxRx.sReceived, ';d:');
		OutputGlobal.Resulth:=MID(fbTCP.TxRx.sReceived,TempPos2-(TempPos1+3),TempPos1+3);
		
		TempPos1:=FIND(fbTCP.TxRx.sReceived, ';d:');
		TempPos2:=FIND(fbTCP.TxRx.sReceived, ';b1:');
		OutputGlobal.Resultd:=MID(fbTCP.TxRx.sReceived,TempPos2-(TempPos1+3),TempPos1+3);
		
		//extract Bool 
		TempPos1:=FIND(fbTCP.TxRx.sReceived, ';b1:');
		OutputGlobal.Boole:=STRING_TO_INT(MID(fbTCP.TxRx.sReceived,1,TempPos1+4));
		
		TempPos1:=FIND(fbTCP.TxRx.sReceived, ';b2:');
		OutputGlobal.Boolh:=STRING_TO_INT(MID(fbTCP.TxRx.sReceived,1,TempPos1+4));
		
		TempPos1:=FIND(fbTCP.TxRx.sReceived, ';b3:');
		OutputGlobal.Boold:=STRING_TO_INT(MID(fbTCP.TxRx.sReceived,1,TempPos1+4));
	END_IF
	
END_IF
END_METHOD

METHOD PUBLIC mConnect
VAR_INPUT

END_VAR
VAR
	
	
END_VAR
//Detecting Rising and falling edge of xEnable and nBusyConnect
REdge(CLK:=xEnable);
FEdge(CLK:=xEnable);
FEdgeBusyConnect(CLK:=fbConnect.bBusy);

//when there is a falling edge on xEnable do a normal déconnection
fbDisconnect.tTimeout:=TCPParam.tTimeout;
fbDisconnect.hSocket:=TCPParam.hSocket;
fbDisconnect.sSrvNetId:=TCPPAram.NetID;
fbDisconnect.bExecute:=FEdge.Q;
fbDisconnect();
OutputDisconnect.xBusy:=fbDisconnect.bBusy;
//TODO: Issue #1
//OutputDisconnect.xError:=fbDisconnect.bError;
OutputDisconnect.nErrID:=403; //TODO: use the errors provided by the FB: Issue #2
IF (FEdge.Q) THEN
	TCPParam.xConnected:=FALSE;
	TCPParam.xConnectedCognex:=FALSE;
	iCounter:=0;
	TCPParam.hSocket.handle:=0;
END_IF

//force disconnecting when xForceDisconnect
fbDisconnectAll.bExecute:=xForceDisconnect;
fbDisconnectAll.tTimeout:=TCPParam.tTimeout;
fbDisconnectAll.sSrvNetId:=TCPPAram.NetID;
fbDisconnectAll();
OutputDisconnectAll.xBusy:=fbDisconnectAll.bBusy;
OutputDisconnectAll.xError:=fbDisconnectAll.bError;
OutputDisconnectAll.nErrID:=403;	//TODO: use the errors provided by the FB: Issue #2
IF (xForceDisconnect) THEN
	TCPParam.xConnected:=FALSE;
	xForceDisconnect:=FALSE;
	xEnable:=FALSE;
	TCPParam.xConnectedCognex:=FALSE;
	iCounter:=0;
	TCPParam.hSocket.handle:=0;
	xReceiveToFast:=FALSE;
END_IF

//Connect to the Server
fbConnect.nRemotePort:=TCPPAram.nRemotePort;
fbConnect.sSrvNetId:=TCPParam.NetID;
fbConnect.sRemoteHost:=TCPParam.sRemoteHost;
fbConnect.tTimeout:=TCPPAram.tTimeout;
fbConnect.bExecute:=REdge.Q;
fbConnect();
OutputConnect.xBusy:=fbConnect.bBusy;
OutputConnect.xError:=fbConnect.bError;
OutputConnect.nErrID:=403;	//TODO: use the errors provided by the FB: Issue #2

IF FEdgeBusyConnect.Q AND fbConnect.hSocket.handle <> 0 THEN
	TCPParam.xConnected:=TRUE;
	TCPParam.xConnectedCognex:=FALSE;
	TCPParam.hSocket:=fbConnect.hSocket;
	iCounter:=0;
	xReceiveToFast:=FALSE;
END_IF
END_METHOD

METHOD PUBLIC mReceive
//Receive data / check for new data each 250mS
Timer.PT:=T#250MS;
//Timer should only work if TCP is currently connected
Timer(IN:=TCPParam.xConnected);

IF (Timer.Q) THEN
	Timer(IN:=FALSE);
	fbReceive.tTimeout:=TCPPAram.tTimeout;
	fbReceive.sSrvNetId:=TCPPAram.NetID;
	fbReceive.cbLen:=200;
	fbReceive.hSocket:=TCPParam.hSocket;
	fbReceive.bExecute:=TRUE;
	fbReceive.pDest:=ADR(sReceivedBuffer);
	IF fbReceive.nRecBytes>0 THEN  //some data received
		IF (TxRx.sReceived='') THEN
			xReceiveToFast:=FALSE;
			TxRx.sReceived:=LEFT(STR:=sReceivedBuffer,SIZE:=UDINT_TO_INT(fbReceive.nRecBytes-2));
		ELSE
			xReceiveToFast:=FALSE;  (*TODO: Set this to true again*)
		END_IF
	END_IF	
ELSE
	fbReceive.bExecute:=FALSE;
END_IF
fbReceive();

//******************************************
//Output actions
//******************************************

OutputReceive.xBusy:=fbReceive.bBusy;
IF xReceiveToFast THEN
	OutputReceive.xError:=TRUE;
	OutputReceive.nErrID:=401;	//TODO: use the errors provided by the FB: Issue #2
ELSE
	OutputReceive.xError:=fbReceive.bError;
	OutputReceive.nErrID:=404;	//TODO: use the errors provided by the FB: Issue #2
END_IF
END_METHOD

METHOD PUBLIC mSend
VAR_INPUT

END_VAR
VAR

END_VAR
IF(TCPParam.xConnected) THEN //only sending when connected
	//Send data when there is something to Send
	fbSend.cbLen:=INT_TO_UINT(LEN(CONCAT(TxRx.sSend,'$R$L')));
	IF(fbSend.cbLen>2 OR fbSend.bBusy) THEN
		IF TxRx.sSend='$R$L' THEN
			fbsend.cbLen:=4;	//only send an "Enter"
		ELSE
			TxRx.sSend:=CONCAT(TxRx.sSend,'$R$L'); //send a whole message
		END_IF
		fbSend.pSrc:=ADR(TxRx.sSend);
		fbSend.sSrvNetId:=TCPPAram.NetID;
		fbSend.hSocket:=TCPParam.hSocket;
		fbSend.tTimeout:=TCPParam.tTimeout;
		fbSend.bExecute:=TRUE;
	END_IF
	fbRTrig(CLK:=fbSend.bBusy);
	IF (fbRTrig.Q) THEN
		fbSend.bExecute:=FALSE;
		TxRx.sSend:='';
	END_IF
	fbSend();
	
	//******************************************
	//Output actions
	//******************************************
	
	OutputSend.xBusy:=fbSend.bBusy;
	OutputSend.xError:=fbSend.bError;
	OutputSend.nErrID:=402;	//TODO: use the errors provided by the FB: Issue #2
	
END_IF
END_METHOD

END_FUNCTION_BLOCK

// ---- ErrorList.TcTLO
TEXTLIST ErrorList
  0 = 'no error' | de: 'kein Fehler' | fr: 'pas de Erreur'
  100 = 'Actuator | Autorisation refused for action Go Out' | de: 'Aktor | Keine Autorisation zum ausfahren' | fr: 'Actionneur | Pas de autorisation pour étendre'
  101 = 'Actuator | Autorisation refused for action Go In' | de: 'Aktor | Keine Autorisation zum einfahren' | fr: 'Actionneur | Pas de autorisation pour retracter'
  110 = 'Actuator | Error timeout go-out' | de: 'Aktor | Timeout ausfahren' | fr: 'Actionneur | Timeout  étendre'
  111 = 'Actuator | Error timeout go-in' | de: 'Aktor | Timeout einfahren' | fr: 'Actionneur | Timeout retracter'
  120 = 'Actuator | Both sensors (IxSensIn & IxSensOut) at the same time' | de: 'Aktor | Beide Sensoren sind gleichzeitig aktiv' | fr: 'Actionneur | Les deux capteurs sont vrai en meme temps'
  121 = 'Actuator | Where shall I go? xSetSort=1 et xSetRentre=1' | de: 'Aktor | Was soll ich tun? xSetSort=1 und xSetRentre=1' | fr: 'Actionneur | Sortir ou rentrer? xSetSort=1 et xSetRentre=1'
  200 = 'Auto | Vision | Error while detecting original object' | de: 'Auto | Vision | Fehler beim Erkennen des Start-Objektes' | fr: "Auto | Vision | Erreur detecter l'object de départ"
  210 = 'Auto | Timeout - Motor did not reach desired speed' | de: 'Auto | Timeout - Motor hat nicht schnell genug den Soll-Wert erreicht' | fr: 'Auto | Timeout - Moteur a pas atteint la vitesse de consigne assez rapide'
  201 = 'Auto | Vision | Error detecting processed object' | de: 'Auto | Vision | Fehler beim Erkennen des End-Objektes' | fr: 'Auto | Vision | Erreur detecter object de fin'
  300 = 'fbMotor | Error in PID-Loop' | de: 'fbMotor | Fehler in der PID-Schleife' | fr: 'fbMotor | Erreur dans boucle PID'
  301 = 'fbMotor | Unable to reach Setpoint Speed' | de: 'fbMotor | Kann Setpoint-Wert nicht erreichen' | fr: "fbMoteur | Impossible d'atteindre la vitesse de consigne"
  401 = 'fbTCP | mReceive | Received Data was lost' | de: 'fbTCP | mReceive | Verlust von eingehenden Daten ' | fr: 'fbTCP | mReceive | Perte de donnes en entree'
  402 = 'fbTCP | Error sending data' | de: 'fbTCP | Fehler beim Senden der Daten' | fr: "fbTCP | Probleme lorsque de l'envoi des données"
  403 = 'fbTCP | Error connecting /disconnecting to Server' | de: 'fbTCP | Fehler beim Verbinden / Trennen der Verbindung zum Server' | fr: 'fbTCP | Erreur lorsque de la (de-)connexion aux Serveur'
  404 = 'fbTCP | mReceive | Error while Receiving data' | de: 'fbTCP | mReceive | Fehler beim Empfangen von Daten' | fr: 'fbTCP | mReceive | Probleme de réception'
  202 = 'Auto | Camera | Error while taking image'
  1 = 'Air Pressure low' | de: 'Luftdruck zu gering' | fr: "Pression d'air trop basse"
   = ''
END_TEXTLIST

// ---- GlobalTextList.TcGTLO
TEXTLIST GlobalTextList
  58 = '%d'
  37 = '%i'
  3 = '%s'
  60 = 'Act1'
  62 = 'Act2'
  61 = 'Act3'
  15 = 'Actionneur 1' | fr: 'Actionneur 1' | de: 'Aktor 1' | en: 'Actuator 1'
  16 = 'Actionneur 2' | fr: 'Actionneur 2' | de: 'Aktor 2' | en: 'Actuator 2'
  17 = 'Actionneur 3' | fr: 'Actionneur 3' | de: 'Aktor 3' | en: 'Actuator 3'
  40 = 'Admin'
  67 = 'ADMIN'
  127 = 'Air pressure emulator'
  8 = 'ARU' | fr: 'ARU' | de: 'NOT-Aus' | en: 'emergency Stop'
  93 = 'ARU - when there is no hardwarebutton present' | fr: 'ARU - seulement si il y a pas de Bouton Hardware' | de: 'NOT-Aus - nur wenn es kein Hardware-Button gibt' | en: 'emergency Stop - only when there is no Hardware Button'
  143 = 'Auto'
  71 = 'AUTOMATIC' | fr: 'AUTOMATIQUE' | de: 'AUTOMATISCH'
  136 = 'Backward'
  126 = 'Camera Control'
  53 = 'Charge' | fr: 'Charge' | de: 'Laden' | en: 'Load'
  96 = 'Connected to Server' | fr: 'Connecté aux Serveur' | de: 'Verbunden mit Serveur'
  25 = 'Consigne: %.2f' | fr: 'Consigne: %.2f' | de: 'Soll-Wert: %.2f' | en: 'Setpoint: %.2f'
  0 = 'Cycle Init' | fr: 'CYCLE INITIALISATION' | de: 'INITIALISIERUNGSZYKLUS' | en: 'INITIALISATION CYCLE'
  5 = 'Cycle Man' | fr: 'CYCLE MANUEL' | de: 'MANUELLER ZYKLUS' | en: 'MANUAL CYCLE'
  92 = 'd: %s'
  63 = 'Direction' | fr: 'Sens de rotation' | de: 'Drehrichtung' | en: 'Direction'
  76 = 'Disable Sensor In - Out' | fr: 'Désactiver Capteur In-Out' | de: 'In-Out Sensor deaktivieren' | en: 'Disable Sensor In-Out'
  114 = 'Do next step if Pas-a-Pas is enabled' | fr: 'Faire le prochain pas si Pas-a-Pas est allumée' | de: 'Nächster Schritt wenn Schritt-für-Schritt aktiviert ist' | en: 'Do next step if Step-for-Step is turned on'
  113 = 'Do Step' | fr: 'Faire un pas' | de: 'Schritt' | en: 'Do Step'
  90 = 'e: %s'
  133 = 'Emulate Z Done'
  97 = 'Enabled' | fr: 'Activé' | de: 'Aktiviert'
  41 = 'english' | fr: 'Anglais' | de: 'Englisch' | en: 'English'
  78 = 'ErrID: %d'
  7 = 'Error' | fr: 'Erreur' | de: 'Fehler' | en: 'Error'
  33 = 'fbConfig.lrTemp : %.2f'
  36 = 'fbConfig.lrValInc : %.2f'
  32 = 'fbConfig.udiNbreIncBus : %i'
  105 = 'fbMotor.fbMotor.fbConvertNumToMotorOut.QaSortie'
  98 = 'Force Disconnect' | de: 'Zwangs-Trennen'
  135 = 'Forward'
  134 = 'ForwardHomePosition'
  19 = 'french' | fr: 'Francais' | de: 'Französisch' | en: 'French'
  43 = 'Gain : %.2f'
  20 = 'german' | fr: 'Allemand' | de: 'Deutsch' | en: 'German'
  65 = 'go back' | fr: 'retour...' | de: 'zurück...' | en: 'go back...'
  66 = 'go back...' | fr: 'retour...' | de: 'zurück...' | en: 'go back...'
  22 = 'Going in' | fr: 'rétracter' | de: 'ein-fahren' | en: 'retract'
  21 = 'Going out' | fr: 'étendre' | de: 'aus-fahren' | en: 'extend'
  91 = 'h: %s'
  128 = 'HomingPos Emulator'
  48 = 'ID: %d'
  142 = 'Init'
  102 = 'Ir Ecart : %.5f'
  103 = 'Ir Tension: %.2f'
  2 = 'LANGUAGE' | fr: 'LANGUE' | de: 'SPRACHE' | en: 'LANGUAGE'
  138 = 'Language'
  140 = 'Language / User'
  115 = 'Login' | fr: 'Connecter' | de: 'Einloggen'
  119 = 'login as another user' | fr: 'Login comme autre utilisateur' | de: 'Als anderen Benutzer einloggen'
  116 = 'Logout' | fr: 'Déconnecter' | de: 'Ausloggen'
  34 = 'lrEcart : %.5f'
  35 = 'lrTension : %.2f'
  4 = 'MAIN' | fr: 'PRINCIPAL' | de: 'HAUPTSEITE' | en: 'MAIN'
  137 = 'Main Speed Control'
  109 = 'MAIN.fbCycleInit.fbEtape.sMess'
  108 = 'MAIN.fbCycleInit.iEtape'
  106 = 'MAIN.fbCycleMan.fbEtape.sMess'
  107 = 'MAIN.fbCycleMan.iEtape'
  139 = 'MainControl'
  144 = 'Manual'
  6 = 'MMA'
  13 = 'Mode Auto'
  12 = 'Mode Init'
  14 = 'Mode Manual'
  112 = 'Mode Pas-a-Pas'
  130 = 'Mot X'
  131 = 'Mot Y'
  129 = 'Mot Z'
  55 = 'Motor' | fr: 'Moteur' | de: 'Motor' | en: 'Motor'
  59 = 'MOTOR' | fr: 'MOTEUR' | de: 'MOTOR' | en: 'MOTOR'
  89 = 'NetID: %s'
  39 = 'None'
  110 = 'Num Output: %d'
  111 = 'Num Output: %i'
  73 = 'Number produced: %d' | fr: 'Nombre produits: %d' | de: 'Anzahl Produziert: %d' | en: 'Number produced: %d'
  75 = 'On            Off'
  68 = 'Open Admin Page' | fr: 'Page administrateur...' | de: 'Admin-Seite' | en: 'Admin Page...'
  64 = 'open more...' | fr: "plus d'info..." | de: 'mehr...' | en: 'open more...'
  46 = 'Operator'
  47 = 'Operator - Service - Admin'
  120 = 'Please login as another user' | fr: 'Veuillez utiliser un autre identifiant' | de: 'Bitte mit anderen Benutzerkennung einloggen'
  104 = 'Qa Sortie : %d'
  101 = 'Qa Sortie : %i'
  38 = 'QaSortie : %2.5f'
  42 = 'QaSortie : %2.5f tr/min'
  31 = 'QaSortie : %i'
  100 = 'QASortie: %i'
  70 = 'Ready' | fr: 'Pret' | de: 'Bereit' | en: 'Ready'
  57 = 'RealSpeed: %d'
  85 = 'Received Data: %s'
  80 = 'Remote IP-Adress: %s'
  81 = 'Remote Port: %d'
  72 = 'Remote Socket: %d'
  10 = 'Rentre       Sort'
  11 = 'Rentre      Sort'
  9 = 'Rentre     Sort'
  49 = 'Reset'
  69 = 'Running' | fr: 'Marche' | de: 'Betrieb' | en: 'Running'
  82 = 'Send Data: %s'
  45 = 'Service'
  132 = 'Set HomePosition'
  1 = 'SetSpeed of Motor: %.2f'
  99 = 'SetSpeed of Motor: %i'
  56 = 'SetSpeed: %d'
  23 = 'Start'
  141 = 'Status'
  148 = 'Status Full'
  147 = 'Status Simple'
  26 = 'stConfigBus.uiNbBits: %i'
  24 = 'Stop'
  27 = 'stTension.lrMax : %.2f'
  28 = 'stTension.lrMin : %.2f'
  29 = 'stValeur.lrMax : %.2f'
  30 = 'stValeur.lrMin : %.2f'
  18 = 'TachoInput: %.2f'
  95 = 'TCP Busy'
  123 = 'TCP Send'
  54 = 'Tighten' | fr: 'Serrage' | de: 'Spannen' | en: 'Tighten'
  125 = 'TRIG    CHECK   GETRES'
  124 = 'TRIG CHECK GETRES'
  117 = 'User'
  121 = 'USER' | fr: 'UTILISATEUR' | de: 'BENUTZER'
  122 = 'User Settings' | fr: 'Param. Utilisateur' | de: 'Benutzer Einst.'
  44 = 'WriteSpeed: %d'
  145 = 'X'
  74 = 'xBusy'
  83 = 'xConnected'
  86 = 'xConnectedCognex'
  94 = 'xConnectedCognex Native'
  51 = 'xEnable'
  87 = 'xEnableCognexMode'
  88 = 'xEnableEmulateTCP'
  77 = 'xError'
  84 = 'xForceDisconnect'
  79 = 'xSend'
  50 = 'xVonnected'
  146 = 'Y'
  118 = 'You are not allowed to see this page' | fr: 'Yous avez pas le droit de voir cette page' | de: 'Sie haben nicht die erforderlichen Recte diese Seite einzusehen'
  52 = 'Z-Axis' | fr: 'Axe Z' | de: 'Z-Achse' | en: 'Z-Axis'
END_TEXTLIST

// ---- VISUs/Visu2_MainCtr.TcVIS
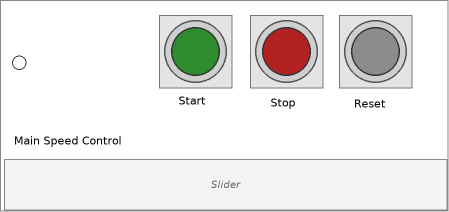
VISUALIZATION Visu2_MainCtr  // 449x212
    Slider (4,159 443x51), variable: stIO.stIn.iSetSpeedMotor, scale 0..100
    RadioButton (10,14 150x97), variable: stParam.stStatus.eMMA
        Areas[0]: Text=Mode Init
        Areas[1]: Text=Mode Auto
        Areas[2]: Text=Mode Manual
    PushSwitch (159,15 73x73), tooltip "Start", variable: stIO.stIn.xStartIO, behaviour: TAP, style: Switch-PushSwitch-Green
    PushSwitch (250,15 73x73), tooltip "Stop", variable: stIO.stIn.xStopIO, invisible if: fbMMA.iEtape<>350, behaviour: TAP, style: Switch-PushSwitch-Red
    PushSwitch (339,15 73x73), tooltip "Reset", variable: stIO.stIn.xResetIO, behaviour: TAP, style: Switch-PushSwitch-Gray
    Label (152,86 80x30), "Start"
    Label (243,88 80x30), "Stop", invisible if: fbMMA.iEtape<>350
    Label (330,89 80x30), "Reset", invisible if: fbMMA.iEtape<>350
    Label (11,126 176x30), "Main Speed Control"
END_VISUALIZATION

// ---- VISUs/Visu2_LanguageUser.TcVIS
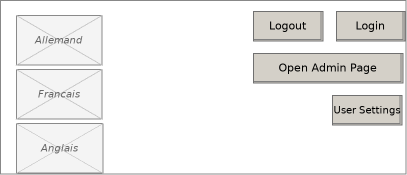
VISUALIZATION Visu2_LanguageUser  // 407x175
    Button (253,53 150x30), "Open Admin Page"
        OnMouseClick: change screen: VisuAdmin
    Button (336,11 69x30), "Login"
        OnMouseClick: VisuUserMgmt Type=Login
    Button (253,11 70x30), "Logout"
        OnMouseClick: VisuUserMgmt Type=Logout
    Button (332,95 70x30), "User Settings"
        OnMouseClick: VisuUserMgmt Type=OpenUserConfiguration
    Image (16,15 86x50), image: Allemand
        OnMouseClick: ChangeLanguage ChangeLanguage=de
    Image (16,69 86x50), image: Francais
        OnMouseClick: ChangeLanguage ChangeLanguage=fr
    Image (16,123 87x50), image: Anglais
        OnMouseClick: ChangeLanguage ChangeLanguage=en
END_VISUALIZATION

// ---- VISUs/Visu2_Status.TcVIS
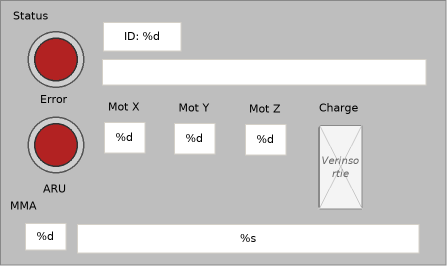
VISUALIZATION Visu2_Status  // 447x266
    Rectangle (-2,-2 447x266)
    Image (318,126 43x83), invisible if: fbAct1.xInInPos=0, image: Verinrentree
    Rectangle (320,150 37x38), "Going out", invisible if: fbAct1.xGoingOutNow=0
    Lamp1 (22,112 68x66), variable: fbBtn.xAru=0, style: Lamp-Lamp1-Red
    Lamp1 (23,25 66x69), variable: stParam.stStatus.xErreur, style: Lamp-Lamp1-Red
    Textfield (102,59 324x26), text variable: stParam.stStatus.sMessage, text list: 'ErrorList', text index: stParam.stStatus.iId
    Textfield (103,22 78x29), "ID: %d", text variable: stParam.stStatus.iId
    Label (299,93 80x30), "Charge"
    Image (319,125 43x84), invisible if: fbAct1.xInOutPos=0, image: Verinsortie
    Textfield (245,124 41x31), "%d", text variable: fbMotorZ.fbAxisRef.NcToPlc.ActPos
    Label (225,94 80x30), "Mot Z"
    Label (154,93 80x30), "Mot Y"
    Textfield (174,123 41x31), "%d", text variable: fbMotorY.fbAxisRef.NcToPlc.ActPos
    Label (84,92 80x30), "Mot X"
    Textfield (104,122 41x31), "%d", text variable: fbMotorX.fbAxisRef.NcToPlc.ActPos
    Label (10,1 176x30), "Status"
    Label (26,85 55x29), "Error"
    Label (11,175 87x28), "ARU"
    Label (7,191 80x30), "MMA"
    Textfield (77,224 342x29), "%s", text variable: fbMMA.fbEtape.sMess
    Textfield (25,223 41x27), "%d", text variable: fbMMA.iEtape
END_VISUALIZATION

// ---- VISUs/Visu2_StatusSimple.TcVIS
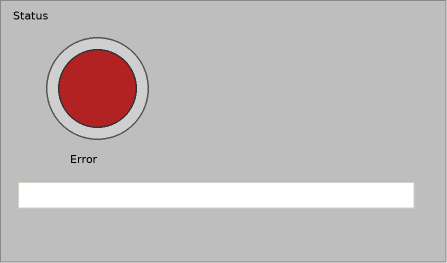
VISUALIZATION Visu2_StatusSimple  // 447x263
    Rectangle (-2,-2 447x263)
    Lamp1 (29,29 137x119), variable: fbBtn.xAru=0 OR stParam.stStatus.xErreur, style: Lamp-Lamp1-Red
    Textfield (18,182 396x26), text variable: stParam.stStatus.sMessage, text list: 'ErrorList', text index: stParam.stStatus.iId
    Label (10,1 176x30), "Status"
    Label (56,145 55x29), "Error"
END_VISUALIZATION

// ---- VISUs/VisuAdmin.TcVIS
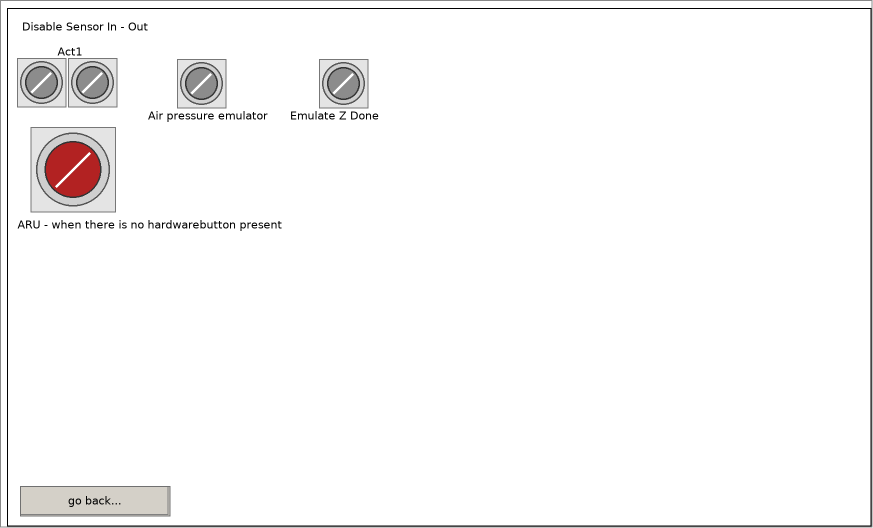
VISUALIZATION VisuAdmin  // 873x528
    Group (265,213 240x84)
        Label (0,0 237x66), "You are not allowed to see this page"
        Label (3,18 237x66), "Please login as another user"
    Rectangle (7,8 864x518)
    Button (20,486 150x30), "go back..."
        OnMouseClick: change screen: Visualization
    Label (-5,37 150x30), "Act1"
    Label (10,12 150x30), "Disable Sensor In - Out"
    RotarySwitch (17,57 49x51), variable: fbAct1.stParam.xPresenceSensIn, behaviour: TOGGLE, style: Switch-RotarySwitch-Gray
    RotarySwitch (68,57 49x51), variable: fbAct1.stParam.xPresenceSensOut, behaviour: TOGGLE, style: Switch-RotarySwitch-Gray
    RotarySwitch (22,127 102x85), variable: stIO.stIn.IxAruIO, behaviour: TOGGLE, style: Switch-RotarySwitch-Red
    Label (1,210 298x30), "ARU - when there is no hardwarebutton present"
    RotarySwitch (177,58 49x51), variable: stio.stIn.xAirPressureOk, behaviour: TOGGLE, style: Switch-RotarySwitch-Gray
    Label (145,101 298x30), "Air pressure emulator"
    Label (287,101 298x30), "Emulate Z Done"
    RotarySwitch (319,58 49x51), variable: stIO.stIn.xEmulateZDone, behaviour: TOGGLE, style: Switch-RotarySwitch-Gray
END_VISUALIZATION

// ---- VISUs/Visualization.TcVIS
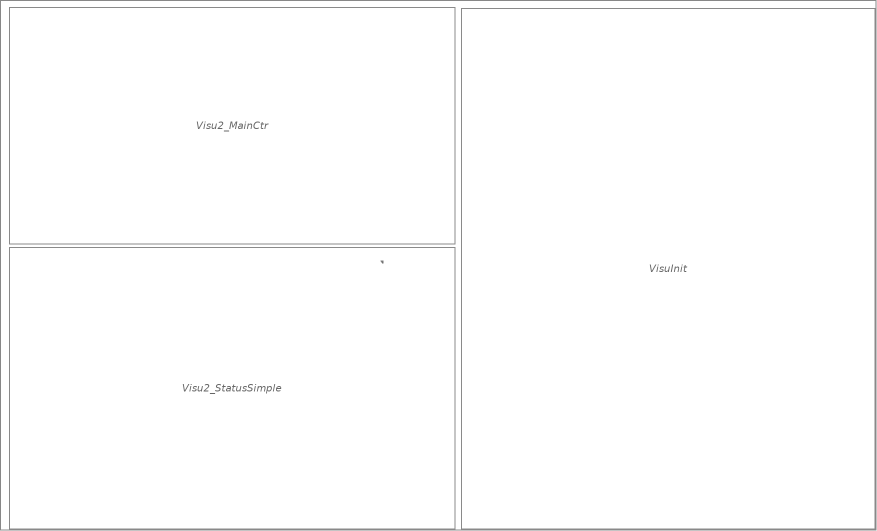
VISUALIZATION Visualization  // 877x531
    Button (382,261 1x2)
    TabControl (9,7 446x237)
        shows Visu2_MainCtr()
        shows Visu2_LanguageUser()
        [0]: TabTitle=MainControl
        [1]: TabTitle=Language / User
    TabControl (461,8 414x521), frame switch variable: stParam.stStatus.eMMA
        shows VisuInit()
        shows VisuAuto()
        shows VisuManual()
        [0]: TabTitle=Init
        [1]: TabTitle=Auto
        [2]: TabTitle=Manual
    TabControl (9,247 446x282)
        shows Visu2_StatusSimple()
        shows Visu2_Status()
        [0]: TabTitle=Status Simple
        [1]: TabTitle=Status Full
END_VISUALIZATION

// ---- VISUs/VisuAuto.TcVIS
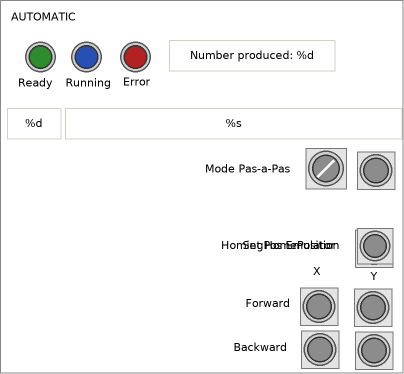
VISUALIZATION VisuAuto  // 404x374
    Label (8,2 116x30), "AUTOMATIC"
    Textfield (65,108 337x31), "%s", text variable: fbCycleAuto.fbEtape.sMess
    Lamp1 (68,39 37x36), variable: fbCycleAuto.xBusy, style: Lamp-Lamp1-Blue
    Label (59,68 59x30), "Running"
    Lamp1 (22,39 37x36), variable: fbCycleAuto.xReady, style: Lamp-Lamp1-Green
    Label (6,68 59x30), "Ready"
    Lamp1 (117,39 37x36), variable: fbCycleAuto.xError, style: Lamp-Lamp1-Red
    Label (107,67 59x30), "Error"
    Textfield (7,108 54x31), "%d", text variable: fbCycleAuto.iEtape
    Textfield (169,40 166x31), "Number produced: %d", text variable: fbCycleAuto.iNumberProduced
    RotarySwitch (305,148 42x41), variable: stParam.stStatus.xModePasAPas, behaviour: TOGGLE, style: Switch-RotarySwitch-Gray
    Label (182,154 111x30), "Mode Pas-a-Pas"
    PushSwitch (357,151 38x39), tooltip "Do next step if Pas-a-Pas is enabled", variable: fbBtn.xNextPas, invisible if: NOT stParam.stStatus.xModePasAPas, behaviour: TAP, style: Switch-PushSwitch-Gray
    Group (194,227 199x145)
        PushSwitch (161,0 38x43), variable: stIO.stIn.xSetHomePos, invisible if: fbCycleInit.iEtape<>500, behaviour: TAP, style: Switch-PushSwitch-Gray
        Label (46,4 102x29), "Set HomePosition", invisible if: fbCycleInit.iEtape<>500
        PushSwitch (106,58 38x43), variable: stIO.stIn.xJogXForward, invisible if: fbCycleInit.iEtape<>500, behaviour: TAP, style: Switch-PushSwitch-Gray
        PushSwitch (161,102 38x43), variable: stIO.stIn.xJogYBackward, invisible if: fbCycleInit.iEtape<>500, behaviour: TAP, style: Switch-PushSwitch-Gray
        PushSwitch (160,59 38x43), variable: stIO.stIn.xJogYForward, invisible if: fbCycleInit.iEtape<>500, behaviour: TAP, style: Switch-PushSwitch-Gray
        PushSwitch (107,101 38x43), variable: stIO.stIn.xJogXBackward, invisible if: fbCycleInit.iEtape<>500, behaviour: TAP, style: Switch-PushSwitch-Gray
        Label (2,62 97x29), "Forward", invisible if: fbCycleInit.iEtape<>500
        Label (0,106 96x29), "Backward", invisible if: fbCycleInit.iEtape<>500
        Label (106,30 34x29), "X", invisible if: fbCycleInit.iEtape<>500
        Label (163,35 34x29), "Y", invisible if: fbCycleInit.iEtape<>500
        Label (5,5 139x27), "HomingPos Emulator", invisible if: stParam.stStatus.xHomingDone
        PushSwitch (163,1 36x36), tooltip "Do next step if Pas-a-Pas is enabled", variable: stIO.stIn.xHomingPosReached, invisible if: stParam.stStatus.xHomingDone, behaviour: TAP, style: Switch-PushSwitch-Gray
END_VISUALIZATION

// ---- VISUs/VisuInit.TcVIS
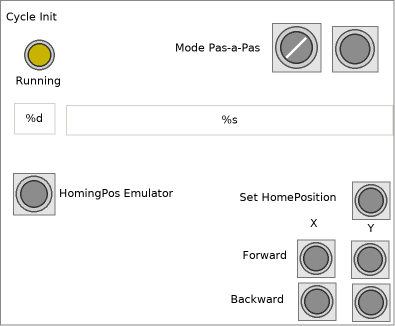
VISUALIZATION VisuInit  // 395x326
    Lamp1 (21,37 37x36), variable: fbCycleInit.xBusy, style: Lamp-Lamp1-Yellow
    Label (3,2 137x30), "Cycle Init"
    Label (9,66 59x30), "Running"
    Textfield (66,105 327x30), "%s", text variable: fbCycleInit.fbEtape.sMess
    Textfield (14,103 41x31), "%d", text variable: fbCycleInit.iEtape
    RotarySwitch (272,22 49x51), variable: stParam.stStatus.xModePasAPas, behaviour: TOGGLE, style: Switch-RotarySwitch-Gray
    Label (152,33 111x30), "Mode Pas-a-Pas"
    PushSwitch (13,173 42x42), tooltip "Do next step if Pas-a-Pas is enabled", variable: stIO.stIn.xHomingPosReached, invisible if: stParam.stStatus.xHomingDone, behaviour: TAP, style: Switch-PushSwitch-Gray
    Label (56,180 139x27), "HomingPos Emulator", invisible if: stParam.stStatus.xHomingDone
    PushSwitch (332,25 46x48), tooltip "Do next step if Pas-a-Pas is enabled", variable: fbBtn.xNextPas, behaviour: TAP, style: Switch-PushSwitch-Gray
    Group (191,179 199x145)
        Label (2,62 97x29), "Forward", invisible if: fbCycleInit.iEtape<>500
        Label (0,106 96x29), "Backward", invisible if: fbCycleInit.iEtape<>500
        Group (46,0 153x145)
            PushSwitch (115,0 38x43), variable: stIO.stIn.xSetHomePos, invisible if: fbCycleInit.iEtape<>500, behaviour: TAP, style: Switch-PushSwitch-Gray
            Label (0,4 102x29), "Set HomePosition", invisible if: fbCycleInit.iEtape<>500
            PushSwitch (60,58 38x43), variable: stIO.stIn.xJogXForward, invisible if: fbCycleInit.iEtape<>500, behaviour: TAP, style: Switch-PushSwitch-Gray
            PushSwitch (115,102 38x43), variable: stIO.stIn.xJogYBackward, invisible if: fbCycleInit.iEtape<>500, behaviour: TAP, style: Switch-PushSwitch-Gray
            PushSwitch (114,59 38x43), variable: stIO.stIn.xJogYForward, invisible if: fbCycleInit.iEtape<>500, behaviour: TAP, style: Switch-PushSwitch-Gray
            PushSwitch (61,101 38x43), variable: stIO.stIn.xJogXBackward, invisible if: fbCycleInit.iEtape<>500, behaviour: TAP, style: Switch-PushSwitch-Gray
            Label (60,30 34x29), "X", invisible if: fbCycleInit.iEtape<>500
            Label (117,35 34x29), "Y", invisible if: fbCycleInit.iEtape<>500
END_VISUALIZATION

// ---- VISUs/VisuManual.TcVIS
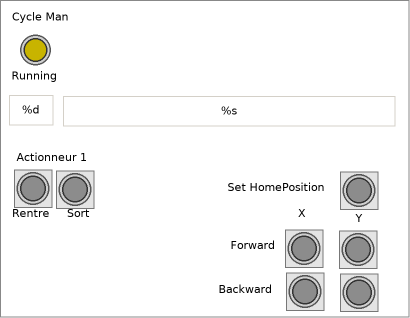
VISUALIZATION VisuManual  // 410x318
    Label (9,2 159x30), "Cycle Man"
    Label (5,61 59x30), "Running"
    Lamp1 (17,32 37x36), variable: fbCycleMan.xBusy, style: Lamp-Lamp1-Yellow
    PushSwitch (14,167 38x43), variable: stIO.stIn.xManualAct1GoIn, behaviour: TAP, style: Switch-PushSwitch-Gray
    PushSwitch (56,168 38x43), variable: stIO.stIn.xManualAct1GoOut, behaviour: TAP, style: Switch-PushSwitch-Gray
    Label (0,199 102x29), "Rentre Sort"
    Label (1,143 102x29), "Actionneur 1"
    Label (306,201 102x29)
    Textfield (63,96 332x30), "%s", text variable: fbCycleMan.fbEtape.sMess
    Textfield (9,95 44x30), "%d", text variable: fbCycleMan.iEtape
    Label (-2,287 155x29)
    Group (179,169 199x145)
        Label (2,62 97x29), "Forward", invisible if: fbCycleInit.iEtape<>500
        Label (0,106 96x29), "Backward", invisible if: fbCycleInit.iEtape<>500
        Group (46,0 153x145)
            PushSwitch (115,0 38x43), variable: stIO.stIn.xSetHomePos, invisible if: fbCycleInit.iEtape<>500, behaviour: TAP, style: Switch-PushSwitch-Gray
            Label (0,4 102x29), "Set HomePosition", invisible if: fbCycleInit.iEtape<>500
            PushSwitch (60,58 38x43), variable: stIO.stIn.xJogXForward, invisible if: fbCycleInit.iEtape<>500, behaviour: TAP, style: Switch-PushSwitch-Gray
            PushSwitch (115,102 38x43), variable: stIO.stIn.xJogYBackward, invisible if: fbCycleInit.iEtape<>500, behaviour: TAP, style: Switch-PushSwitch-Gray
            PushSwitch (114,59 38x43), variable: stIO.stIn.xJogYForward, invisible if: fbCycleInit.iEtape<>500, behaviour: TAP, style: Switch-PushSwitch-Gray
            PushSwitch (61,101 38x43), variable: stIO.stIn.xJogXBackward, invisible if: fbCycleInit.iEtape<>500, behaviour: TAP, style: Switch-PushSwitch-Gray
            Label (60,30 34x29), "X", invisible if: fbCycleInit.iEtape<>500
            Label (117,35 34x29), "Y", invisible if: fbCycleInit.iEtape<>500
END_VISUALIZATION

// ---- VISUs/VisuMMA.TcVIS
VISUALIZATION VisuMMA  // 2x2
END_VISUALIZATION

// ---- VISUs/VisuMotor.TcVIS
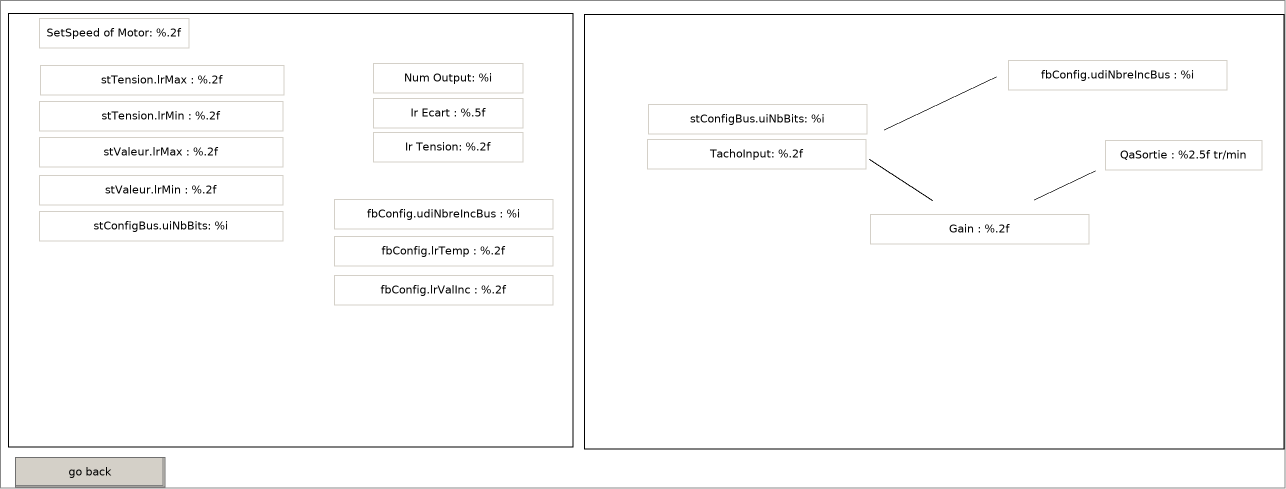
VISUALIZATION VisuMotor  // 1286x489
    Group (160,59 240x84)
        Label (0,0 237x66), "You are not allowed to see this page"
        Label (3,18 237x66), "Please login as another user"
    Rectangle (8,13 565x434)
    Rectangle (584,14 700x435)
    Button (15,457 150x30), "go back", text list: ''
        OnMouseClick: change screen: Visualization
    Line (869,159) (932,200)
    Line (1095,171) (1034,200)
    Line (996,77) (884,130)
    Textfield (373,98 150x30), "Ir Ecart : %.5f", text variable: fbMotor.fbConvertNumToMotorOut.lrEcart
    Textfield (373,132 150x30), "Ir Tension: %.2f", text variable: fbMotor.fbConvertNumToMotorOut.lrTension
    Textfield (40,65 244x30), "stTension.lrMax : %.2f", text variable: fbMotor.fbConvertNumToMotorOut.fbConfig.stTension.lrMax
        OnMouseClick: write the text variable via Default
    Textfield (39,18 150x30), "SetSpeed of Motor: %.2f", text variable: fbMotor.fbConvertNumToMotorOut.lrConsigne
    Textfield (39,101 244x30), "stTension.lrMin : %.2f", text variable: fbMotor.fbConvertNumToMotorOut.fbConfig.stTension.lrMin
        OnMouseClick: write the text variable via Default
    Textfield (39,137 244x30), "stValeur.lrMax : %.2f", text variable: fbMotor.fbConvertNumToMotorOut.fbConfig.stValeur.lrMax
        OnMouseClick: write the text variable via Default
    Textfield (39,175 244x30), "stValeur.lrMin : %.2f", text variable: fbMotor.fbConvertNumToMotorOut.fbConfig.stValeur.lrMin
        OnMouseClick: write the text variable via Default
    Textfield (39,211 244x30), "stConfigBus.uiNbBits: %i", text variable: fbMotor.fbConvertNumToMotorOut.fbConfig.uiNbreBitBus
        OnMouseClick: write the text variable via Default
    Textfield (334,199 219x30), "fbConfig.udiNbreIncBus : %i", text variable: fbMotor.fbConvertNumToMotorOut.fbConfig.udiNbreIncBus
        OnMouseClick: write the text variable via Default
    Textfield (334,236 219x30), "fbConfig.lrTemp : %.2f", text variable: fbMotor.fbConvertNumToMotorOut.fbConfig.lrTemp
        OnMouseClick: write the text variable via Default
    Textfield (334,275 219x30), "fbConfig.lrValInc : %.2f", text variable: fbMotor.fbConvertNumToMotorOut.fbConfig.lrValInc
        OnMouseClick: write the text variable via Default
    Textfield (648,104 219x30), "stConfigBus.uiNbBits: %i", text variable: fbMotor.fbConvertTachoToNumSpeed.fbConfig.uiNbreBitBus
        OnMouseClick: write the text variable via Default
    Textfield (647,139 219x30), "TachoInput: %.2f", text variable: fbMotor.fbConvertTachoToNumSpeed.IaEntree
        OnMouseClick: write the text variable via Default
    Textfield (1105,140 157x30), "QaSortie : %2.5f tr/min", text variable: fbMotor.fbConvertTachoToNumSpeed.lrValeur
        OnMouseClick: write the text variable via Default
    Textfield (870,214 219x30), "Gain : %.2f", text variable: fbMotor.fbConvertTachoToNumSpeed.fbConfig.stValeur.lrMax
        OnMouseClick: write the text variable via Default
    Textfield (1008,60 219x30), "fbConfig.udiNbreIncBus : %i", text variable: fbMotor.fbConvertTachoToNumSpeed.fbConfig.uiNbreBitBus
        OnMouseClick: write the text variable via Default
    Textfield (373,63 150x30), "Num Output: %i", text variable: fbMotor.fbConvertNumToMotorOut.QaSortie
        OnMouseClick: write the text variable via Default
END_VISUALIZATION
